# B&R Automation Studio project 8238 (part 22)

#### CmdSI.typ - BatchInformation / 1002
```iecst
(********************************************************************
 * COPYRIGHT -- Herbert Kannegiesser GmbH
 ********************************************************************
 * Library: Kanlink Cmd 1004 Status Information
 * File: CmdSI.typ
 * Author: Horn
 * Created: 02.03.2016
 ********************************************************************
 * Data types of library Kanlink
 ********************************************************************)
(*Kommando*)

TYPE
	KLreq1004_Status_typ : 	STRUCT
		wCntPositions : UINT;
		wCmdReq : UINT;
		wNoOfPosition : ARRAY[0..11]OF UINT;
	END_STRUCT;
	KLresp1004_Status_typ : 	STRUCT
		wCntPositions : UINT;
		wCmdResp : UINT;
		wNoOfPositions : ARRAY[0..11]OF UINT;
		StatusInfo : ARRAY[0..11]OF StatusInfo_typ;
	END_STRUCT;
	KL_SI_typ : 	STRUCT
		Req : KLreq1004_Status_typ;
		Resp : KLresp1004_Status_typ;
	END_STRUCT;
	StatusInfo_typ : 	STRUCT
		wStatusX : UINT;
		wSubState : UINT;
		wData1 : UINT;
		wData2 : UINT;
	END_STRUCT;
	StatusDataCmd1_typ : 	STRUCT
		wRemainCycleTime : UINT; (*Resttaktzeit bis zum Transfer*)
		wTargetCycleTime : UINT; (*Solltektzeit ohne Verkürzung oder Verlängerung*)
	END_STRUCT;
END_TYPE
```

#### CmdSilo.typ - Exported data types
```iecst
(********************************************************************
 * COPYRIGHT -- Herbert Kannegiesser GmbH
 ********************************************************************
 * Library: Kanlink
 * File: Kanlink.typ
 * Author: stahlhut
 * Created: 20.03.2012
 ********************************************************************
 * Data types of library Kanlink Commando 30010 Silo
 ********************************************************************)
(*Kommandos*)

TYPE
	KLresp30010_SH_typ : 	STRUCT
		MachineNo : STRING[15];
		State : UINT;
		RouteState : ARRAY[1..20]OF UINT;
		WetAccState : ARRAY[1..10]OF UINT;
		WetAccNiveau_mm : ARRAY[1..10]OF UINT;
		WetAccNiveau_rel : ARRAY[1..10]OF UINT;
		WetAccNiveau_Liter : ARRAY[1..10]OF UINT;
		WetAccTemp : ARRAY[1..10]OF UINT;
		WetAccMinLvlOK : ARRAY[1..10]OF UINT;
		WetAccMaxLvlOK : ARRAY[1..10]OF UINT;
	END_STRUCT;
	KLreq30010_SH_typ : 	STRUCT
		MachineNo : STRING[15];
		State : UINT;
		Handshake : BOOL;
		Route : ARRAY[1..20]OF USINT;
		TankTemp : ARRAY[1..10]OF UINT;
	END_STRUCT;
	KL_SiloData_typ : 	STRUCT
		Req : KLreq30010_SH_typ;
		Resp : KLresp30010_SH_typ;
	END_STRUCT;
END_TYPE
```

#### KLInterface.typ - Interfacetypen Kanlink
```iecst
(********************************************************************
 * COPYRIGHT -- Herbert Kannegiesser GmbH
 ********************************************************************
 * Library: Kanlink	 Interface
 * File:
 * Author: stahlhut
 * Created: 20.03.2012
 ********************************************************************
 * Data types of Interface Kanlink
 ********************************************************************)

TYPE
	KL_Key_typ : 	STRUCT
		IP_Key : UDINT;
		CmdKey : UDINT;
	END_STRUCT;
	KL_Parameter_typ : 	STRUCT
		Server : ARRAY[0..HLKANLINK_MAX_SERVERCONNS] OF KL_ServerPar_typ;
		Client : ARRAY[0..HLKANLINK_MAX_CLIENTCONNS] OF KL_ClientPar_typ;
		adrUserTyp : UDINT;
	END_STRUCT;
	KL_ClientPar_typ : 	STRUCT
		Name : STRING[15];
		Adr : UINT;
		Cmd : UINT;
		CmdOpt : UINT; (*Bits 0..3 = Nummer des Clients*)
		Area : UINT;
		CycleTime : UINT;
		sReq : STRING[80];
		sResp : STRING[80];
		AdvMode : BOOL; (*Modus mit dem eine vollständige IP-Adresse eingegeben werden kann*)
		AdrAdvMode : STRING[16]; (*Vollständige IP-Adresse*)
	END_STRUCT;
	KL_ServerPar_typ : 	STRUCT
		Name : STRING[15];
		Adr : UINT;
		Cmd : UINT;
		CmdOpt : UINT; (*Bits 0..3 = Nummer der Verbindung*)
		Area : UINT;
		TimeOut : UINT;
		sReq : STRING[80];
		sResp : STRING[80];
		AdvMode : BOOL; (*Modus mit dem eine vollständige IP-Adresse eingegeben werden kann
oder die Prüfung der IP-Adresse entfällt.*)
		AdrAdvMode : STRING[16]; (*Vollständige IP-Adresse*)
	END_STRUCT;
	IF_ServerOutTyp : 	STRUCT
		xConnected : BOOL;
		iCfgState : UINT; (*0 = ConfOK*)
		tag : UDINT;
	END_STRUCT;
	IF_Server_typ : 	STRUCT
		iState : UINT;
		out : IF_ServerOutTyp;
		tag : UDINT;
	END_STRUCT;
	IF_ClientOut_typ : 	STRUCT
		xConnected : BOOL;
		recTag : UDINT;
	END_STRUCT;
	IF_Client_typ : 	STRUCT
		out : IF_ClientOut_typ;
		iState : UINT;
		tag : UDINT;
	END_STRUCT;
	IFhlKanLink_Typ : 	STRUCT
		in : IF_KL_Control_in_typ;
		out : IF_KL_Control_out_typ;
		Server : ARRAY[0..HLKANLINK_MAX_SERVERCONNS] OF IF_Server_typ;
		Client : ARRAY[0..HLKANLINK_MAX_CLIENTCONNS] OF IF_Client_typ;
		Parameter : KL_Parameter_typ;
		xError : BOOL; (*Kanlink in Störung*)
	END_STRUCT;
	IF_KL_Control_in_typ : 	STRUCT
		xRun : BOOL; (*Rise= Starten Kanlink /fall = stoppen Kanlink*)
		xRestart : BOOL;
	END_STRUCT;
	IF_KL_Control_out_typ : 	STRUCT
		iError : UINT;
		iServerError : ARRAY[0..HLKANLINK_MAX_SERVERCONNS] OF UINT;
		iClientError : ARRAY[0..HLKANLINK_MAX_CLIENTCONNS] OF UINT;
		iStep : UINT; (*Statemachine KanLink*)
	END_STRUCT;
	IFhlKLVisuIN_typ : 	STRUCT
		cmdNr : INT; (*Ausführbares Commando*)
		cmdTag : INT; (*Dazugehörige Daten*)
		iServerNr : UINT; (*zu lesende Serverlist*)
		iCltNr : UINT; (*zu lesender Client*)
	END_STRUCT;
	IFhlKLVisuOUT_typ : 	STRUCT
		step : UINT;
		udpOpenStatus : UINT;
		udpSendStatus : UINT;
		udpRecStatus : UINT;
		iCycleTime : UINT;
		udNetId : UDINT;
		server : KL_ServerListe_typ;
		client : KL_ClientListe_typ;
		cmdResp : INT; (*Response auf CmdNr*)
	END_STRUCT;
	IFhlKLVisu_typ : 	STRUCT
		in : IFhlKLVisuIN_typ;
		out : IFhlKLVisuOUT_typ;
	END_STRUCT;
END_TYPE
```

#### KanLinkLib.typ - Exported data types
```iecst
(********************************************************************
 * COPYRIGHT -- Herbert Kannegiesser GmbH
 ********************************************************************
 * Library: WetLinkLib
 * File: WetLinkLib.typ
 * Author: stahlhut
 * Created: January 06, 2012
 ********************************************************************
 * Data types of library WetLinkLib
 ********************************************************************)
(*Interne Strukturen*)

TYPE
	udp_typ : 	STRUCT  (*UDP Typ*)
		open : UdpOpen;
		send : UdpSend;
		rec : UdpRecv;
		close : UdpClose;
	END_STRUCT;
	udint_array_typ : 	STRUCT  (*Casten von UDINT -> byte*)
		a : USINT;
		b : USINT;
		c : USINT;
		d : USINT;
	END_STRUCT;
	ServerDataTyp : 	STRUCT  (*Datatyp for global Variables*)
		receive_data : ARRAY[0..8191]OF USINT; (*Data which has been received*)
		send_data : ARRAY[0..8191]OF USINT; (*Data which should be sent*)
		PreHeaderSend : PreHeader_Typ;
		PreHeaderRec : PreHeader_Typ;
		HeaderV1Send : ARRAY[0..KLLIB_MAX_MUL]OF HeaderV1_Typ;
		HeaderV1Rec : ARRAY[0..KLLIB_MAX_MUL]OF HeaderV1_Typ;
		MetaInfoResp : KLresp0_MetaInfo_typ;
		ErrorFrame : KL_Error_Frame_typ;
		PingReq : KLreq2_Ping_typ;
		PingResp : KLresp2_Ping_typ;
		IPAdr : STRING[16]; (*IP-Adresse des Clients*)
	END_STRUCT;
	PreHeader_Typ : 	STRUCT
		Magic : UDINT; (*MagicNr*)
		HeaderVersion : UINT; (*Headerversion*)
		Tag : UINT; (*Reserve*)
	END_STRUCT;
	HeaderV1_Typ : 	STRUCT
		ReqID : UINT;
		dataFormat : UINT;
		Command : UINT;
		Length : UINT;
		CmdNr : UINT;
		CmdTag : UINT; (*Unterschiedliche Parameter zum Command*)
		Tag : UDINT; (*Reserve/Spezial*)
	END_STRUCT;
	KL_ServerListe_typ : 	STRUCT
		Cmd : UINT;
		CmdOpt : UINT;
		Adr : UINT;
		Area : UINT;
		pRespStr : UDINT; (*Adresse des Resp String*)
		pReqStr : UDINT; (*Adresse des Req String*)
		AdrDataReq : UDINT;
		ReqLength : UDINT; (*Länge Request Daten*)
		AdrDataResp : UDINT;
		RespLength : UDINT; (*Länge Response Daten*)
		Key : KL_Key_typ; (*Suchschlüssel/ Darf nicht doppelt vorkommen== Konfigurierungsfehler*)
		xConnected : BOOL; (*Falls Commando 2s nicht angefragt wird ist verbindung unterbrochen*)
		iConnectionTimer : UINT; (*Der Zugehörige Zähler / Timer*)
		adrParameter : UDINT; (*Adresse der Parameter*)
		sServerIPAdr : STRING[16];
		sClientIPAdr : STRING[16];
		iReqCnt : UINT;
		xReqManually : BOOL;
		iReqID : UINT;
		iCfgStatus : UINT;
		adrInterface : UDINT;
		xActiv : BOOL;
		tag : UDINT;
	END_STRUCT;
	KL_MuServerListe_typ : 	STRUCT
		Servers : ARRAY[0..KLLIB_MAX_MUL]OF INT;
		wOffset : ARRAY[0..KLLIB_MAX_MUL]OF UINT;
		MuServer : ARRAY[0..KLLIB_MAX_MUL]OF INT;
		lRespLength : ARRAY[0..KLLIB_MAX_MUL]OF UDINT;
		AdrRespData : ARRAY[0..KLLIB_MAX_MUL]OF UDINT;
		RespData : ARRAY[0..8191]OF USINT; (*Data which should be sent*)
		bMuServerIdx : USINT;
	END_STRUCT;
	KL_MuClientListe_typ : 	STRUCT
		bUse : USINT; (*1 = Multiclient aktiv, 2 = Multiclient wurde noch nicht geprüft, 255 = Server akzeptiert kein Multiclient*)
		Clients : ARRAY[0..KLLIB_MAX_MUL]OF INT;
		sClientAdr : STRING[16];
		iCycleTime : UINT;
		iCnt : UINT;
		iReqId : UINT;
		TimeOut : UINT;
		iTimeOutCnt : UINT;
		iCycleWait : UINT;
		xReqPending : BOOL;
		xActiv : BOOL;
		iTimeOutCnt_Summe : UINT;
		TimeOutLeft : UINT;
		xConnected : BOOL; (*True wenn Verbindung aktiv und läuft*)
		Length : UINT;
		RespLength : UDINT;
		ReqLength : UDINT;
	END_STRUCT;
	KL_ClientListe_typ : 	STRUCT
		RecCmd : UINT; (*Rec Command nr*)
		Cmd : UINT; (*Send Command nr*)
		CmdOpt : UINT; (*SendeOptionen Senden Nr des Commando etc*)
		Adr : UINT;
		Area : UINT;
		Key : KL_Key_typ;
		pResp : UDINT; (*Adresse des Namen der Response Struktur*)
		pReq : UDINT; (*Adresse des Namen der Request Struktur*)
		AdrDataReq : UDINT;
		AdrDataResp : UDINT;
		ReqLength : UDINT;
		RespLength : UDINT;
		TimeOut : UINT;
		TimeOutLeft : UINT;
		xError : BOOL;
		iCycleWait : UINT;
		iCycleTime : UINT;
		xDataRec : BOOL;
		MuClient : SINT; (*Enthalten im Multiclient*)
		iReqId : UINT;
		sClientAdr : STRING[16];
		xReqPending : BOOL;
		iTimeOutCnt : UINT;
		xActiv : BOOL;
		iCnt : UINT;
		xConnected : BOOL; (*True wenn Verbindung aktiv und läuft*)
		iTimeOutCnt_Summe : UINT;
		adrInterface : UDINT;
		adrParameter : UDINT; (*Adresse der Parameter*)
		recTag : UDINT; (*Tag des Kommandos*)
	END_STRUCT;
END_TYPE

(*Kommandos*)

TYPE
	KL_Error_Frame_typ : 	STRUCT
		Version : UINT;
		ErrorNumber : UINT;
		ErrorText : STRING[63];
	END_STRUCT;
	KLresp0_MetaInfo_typ : 	STRUCT
		KanLink_Hostname : STRING[15];
		Machine_type : STRING[15];
		SoftwareNo : STRING[15];
		SoftwareVersion : STRING[15];
		DataModelTimeStamp : DATE_AND_TIME;
		DataModelVersion : UINT;
		TimeZone : UINT;
		SommerTime : UINT;
	END_STRUCT;
	KLreq2_Ping_typ : 	STRUCT
		KanLink_Hostname : STRING[15];
	END_STRUCT;
	KLresp2_Ping_typ : 	STRUCT
		KanLink_Hostname : STRING[15];
		FrameVersion : USINT;
	END_STRUCT;
	BatchData_typ : 	STRUCT
		dtTimeStamp : DATE_AND_TIME;
		bTypeBatchNo : USINT;
		bCntCustomers : USINT;
		wTotalWeight : UINT;
		bBatchNo : ARRAY[0..15]OF USINT;
		sCategory : STRING[11];
		utfMark : ARRAY[0..31]OF UINT;
		bCustom : ARRAY[0..11]OF USINT;
		PartBatch : ARRAY[0..7]OF PartBatchData_typ;
	END_STRUCT;
	PartBatchData_typ : 	STRUCT
		sCustomNo : STRING[11];
		wCustomWeight : UINT;
	END_STRUCT;
END_TYPE
```

#### KanLinkLib.var - Exported constants
```iecst
(********************************************************************
 * COPYRIGHT -- Herbert Kannegiesser GmbH
 ********************************************************************
 * Library: WetLinkLib
 * File: WetLinkLib.var
 * Author: stahlhut
 * Created: January 06, 2012
 ********************************************************************
 * Constants of library WetLinkLib
 ********************************************************************)
VAR CONSTANT
	KLLIB_REQ : USINT := 1;
	KLLIB_MAX_MUL : USINT := 15; (*Maximale Anzahl an Clients die zusammengefasst werden dürfen*)
	KLLIB_RESP : USINT := 2;
	MagicNr : UDINT := 16#B16B00B5;
	PreHeaderSize : UDINT := 8;
	HeaderSize : UDINT := 16;
	KL_optReqManually : UINT := 16#8000;
	KL_optOnReqCall : UINT := 16#4000;
	KLLIB_MSG_NULL_POINTER : UINT := 60000;
	KLLIB_MSG_NOT_ENOUGH_MEM : UINT := 60001;
	KLLIB_MSG_VAR_ERROR : UINT := 60002;
END_VAR
```

#### KanLinkLib.fun - Exported functions and function blocks
```iecst
(********************************************************************
 * COPYRIGHT -- Herbert Kannegiesser GmbH
 ********************************************************************
 * Library: WetLinkLib
 * File: WetLinkLib.fun
 * Author: stahlhut
 * Created: January 06, 2012
 ********************************************************************
 * Functions and function blocks of library WetLinkLib
 ********************************************************************)

FUNCTION_BLOCK KanLink_FB (*TODO: Add your comment here*)
	VAR_INPUT
		Step : UINT; (*state machine*)
		ErrorNr : UINT;
		client_address : STRING[16]; (*Speichern der Receiver Adresse*)
		RecKey : KL_Key_typ;
		sNetID : STRING[15];
		udNetID : UDINT;
		udp : udp_typ;
		ServerData : ServerDataTyp;
		ServerListe : ARRAY[0..HLKANLINK_MAX_SERVERCONNS] OF KL_ServerListe_typ; (*Erlaubte Daten Server*)
		ClientListe : ARRAY[0..HLKANLINK_MAX_CLIENTCONNS] OF KL_ClientListe_typ;
		MuClientListe : ARRAY[0..HLKANLINK_MAX_MU_CLIENTCONNS] OF KL_MuClientListe_typ; (*Zusammenfasseb mehrere Clients in ein Telegramm*)
		MuServerListe : KL_MuServerListe_typ;
		_xOpenPort : BOOL;
		_xSendClient : BOOL;
		_xGetClientResp : BOOL;
		_xGetServerReq : BOOL;
		_uiLastId : UDINT;
		CanReturn : BOOL;
		adrSelf : UDINT; (*Eigene Adresse, zum weiterleiten an Function/Function Block*)
		_offset : UDINT; (*Offset zum Berechnen der Sendelänge*)
		_SendLen : UDINT; (*Sendelänge*)
		DoCommand : UINT;
		KLLib_Init_0 : KLLib_Init;
		_iCycleTime : UINT;
		adrInterface : UDINT;
		iPort : UINT; (*Port nr (23500)*)
		sIF : STRING[10]; (*Interface Ethernet*)
		CfgClient : KLLib_CfgClient;
		CfgServer : KLLib_CfgServer;
	END_VAR
	VAR_OUTPUT
		xReturn : BOOL;
	END_VAR
	VAR
		_dPrehead : REFERENCE TO PreHeader_Typ;
		_dHead : REFERENCE TO HeaderV1_Typ;
		_udArr : REFERENCE TO udint_array_typ;
		_dRecAdr : UDINT;
		_xPreheadOK : BOOL;
		_xVersionOK : BOOL;
		_xUse : BOOL;
		_i : USINT;
	END_VAR
END_FUNCTION_BLOCK

FUNCTION KLLib_ClientTimer : BOOL (*Bearbeitet Timeout und Cycletime (Zähler)*)
	VAR_INPUT
		Srv : REFERENCE TO KanLink_FB;
		_iCycleTime : UINT;
	END_VAR
	VAR
		_dClient : REFERENCE TO KL_ClientListe_typ;
		_k : UINT;
		_i : UINT;
		_dServer : REFERENCE TO KL_ServerListe_typ;
		_dInterface : REFERENCE TO IF_Client_typ;
		_dSrvIf : REFERENCE TO IF_Server_typ;
	END_VAR
END_FUNCTION

FUNCTION KLLib_GetPVAdr : UDINT (*Adresse der PV ermitteln (Server)*)
	VAR_INPUT
		ServerItem : REFERENCE TO KL_ServerListe_typ;
	END_VAR
	VAR
		iStat : INT;
	END_VAR
END_FUNCTION

FUNCTION KLLib_SendData : UDINT (*TODO: Add your comment here*)
	VAR_INPUT
		Srv : REFERENCE TO KanLink_FB;
		SendAdr : UDINT;
		SendLen : UDINT;
		pDestination : UDINT; (*Adresse des Zielstrings*)
		iIndex : INT; (*Alternativ kann zu den SendAdr und der Sende Lenge auch die Instanz des Clients angegeben werden*)
		iMuIndex : INT; (*Bei einem Multiclient wird die SendAdr und die Sende Lenge nicht angegeben.*)
		bMode : USINT; (*0 = Client; 1 = Server // Wird nur angegeben, wenn nicht die direkten Adressen angegeben werden.*)
	END_VAR
	VAR
		_i : USINT;
	END_VAR
END_FUNCTION

FUNCTION KLLib_ReadServerPara : UDINT (*TODO: Add your comment here*)
	VAR_INPUT
		adrServerItem : UDINT;
		adrParaItem : UDINT;
		adrKanLink : UDINT;
	END_VAR
	VAR
		_xError : BOOL;
		KanLink : REFERENCE TO KanLink_FB;
		dServer : REFERENCE TO KL_ServerListe_typ;
		dPara : REFERENCE TO KL_ServerPar_typ;
		_udAdr : UDINT;
		_udArr : REFERENCE TO udint_array_typ;
		_udNetId : REFERENCE TO udint_array_typ;
	END_VAR
END_FUNCTION

FUNCTION KLLib_ReadClientPara : UDINT (*TODO: Add your comment here*)
	VAR_INPUT
		adrClientItem : UDINT;
		adrParaItem : UDINT;
		adrServer : UDINT;
	END_VAR
	VAR
		_xError : BOOL;
		dClient : REFERENCE TO KL_ClientListe_typ;
		dPara : REFERENCE TO KL_ClientPar_typ;
		_udArr : REFERENCE TO udint_array_typ;
		_udAdr : UDINT;
		dServer : REFERENCE TO KanLink_FB;
		_udNetId : REFERENCE TO udint_array_typ;
	END_VAR
END_FUNCTION

FUNCTION KLLib_InitCltPV : UDINT (*TODO: Add your comment here*)
	VAR_INPUT
		dclt : REFERENCE TO KL_ClientListe_typ;
	END_VAR
	VAR
		iStat : UINT;
	END_VAR
END_FUNCTION

FUNCTION_BLOCK KLLib_Init (*TODO: Add your comment here*)
	VAR_INPUT
		enable : BOOL;
		adrServer : UDINT;
		adrInterface : UDINT;
	END_VAR
	VAR_OUTPUT
		status : UINT;
	END_VAR
	VAR
		_bStep : INT;
		_dServer : REFERENCE TO KanLink_FB;
		GetEthPort_0 : kgGetEthPort;
		CfgGetIPAddr_0 : CfgGetIPAddr;
		RTInfo_0 : RTInfo;
		_i : INT;
		_k : INT;
		_m : INT;
		_n : INT;
		_dIf : REFERENCE TO IFhlKanLink_Typ;
	END_VAR
END_FUNCTION_BLOCK

FUNCTION KL_BuildKey : BOOL
	VAR_INPUT
		Command : UINT;
		CmdNr : USINT;
		IPAdr : STRING[16];
		adrKey : UDINT;
	END_VAR
	VAR
		IP_Key : UDINT;
		Key : REFERENCE TO KL_Key_typ;
	END_VAR
END_FUNCTION

FUNCTION_BLOCK KLLib_CfgClient (*Configuriert einen Kanlink Client*)
	VAR_INPUT
		adrKanlink : UDINT;
		ClientIndex : UINT;
		adrName : UDINT;
		IPAdr : USINT;
		Area : USINT;
		CmdOpt : UINT;
		Cmd : UINT;
		CycleTime : UINT;
		adrSReq : UDINT;
		adrSResp : UDINT;
	END_VAR
	VAR_OUTPUT
		status : UINT;
	END_VAR
	VAR
		_dKL : REFERENCE TO KanLink_FB;
		_dCltPar : REFERENCE TO KL_ClientPar_typ;
		_iret : UDINT;
	END_VAR
END_FUNCTION_BLOCK

FUNCTION_BLOCK KLLib_CfgServer (*Configuriert einen Kanlink Server*)
	VAR_INPUT
		adrKanlink : UDINT;
		ServerIndex : UINT;
		adrName : UDINT;
		IPAdr : USINT;
		Area : USINT;
		CmdOpt : UINT;
		Cmd : UINT;
		TimeOut : UINT;
		adrSReq : UDINT;
		adrSResp : UDINT;
	END_VAR
	VAR_OUTPUT
		status : UINT;
	END_VAR
	VAR
		_dKL : REFERENCE TO KanLink_FB;
		_dSrvPar : REFERENCE TO KL_ServerPar_typ;
		_iret : UDINT;
	END_VAR
END_FUNCTION_BLOCK

FUNCTION KLLib_CreateStrucDef : UINT (*Erzeuge eine Strukturdefinition zu einer Variablen*)
	VAR_INPUT
		lPtrAdr : UDINT;
		lPtrLen : UDINT;
		sRootName : STRING[127];
		sItemName : STRING[31];
		lDataAdr : UDINT;
	END_VAR
	VAR
		_wStatus : UINT;
		_sPvName : STRING[127];
		_lDataType : UDINT;
		_lDataLen : UDINT;
		_wDataDimension : UINT;
		_sLine : STRING[127];
		_sValueLen : STRING[11];
		_lAdr : REFERENCE TO UDINT;
		_lLen : REFERENCE TO UDINT;
		_sValueDim : STRING[5];
		_sValueOffs : STRING[11];
		_i : UINT;
		_sItemName : STRING[31];
		_sType : ARRAY[1..23] OF STRING[15] := ['BOOL','SINT','INT','DINT','USINT','UINT','UDINT','REAL','STRING','ULINT','DATE_AND_TIME','TIME','DATE','LREAL','','TIME_OF_DAY','BYTE','WORD','DWORD','LWORD','WSTRING','','LINT'];
		_lDataAdr : UDINT;
	END_VAR
END_FUNCTION

FUNCTION KLLib_WriteStrucDefLine : UINT (*Übertrage einen String als Zeile in den Speicher*)
	VAR_INPUT
		lPtrLine : UDINT;
		lPtrAdr : UDINT;
		lPtrLen : UDINT;
	END_VAR
	VAR
		_lAdr : REFERENCE TO UDINT;
		_lLen : REFERENCE TO UDINT;
		_iStringlen : INT;
		_sLine : REFERENCE TO STRING[127];
	END_VAR
END_FUNCTION
```

#### KLLib_CfgClient.st - Configuriert einen Kanlink Client
```iecst
(********************************************************************
 * COPYRIGHT -- Herbert Kannegiesser GmbH
 ********************************************************************
 * Library: KanLinkLib
 * File: KLLib_CfgServer.st
 * Author: stahlhut
 * Created: February 01, 2012
 ********************************************************************
 * Implementation of library KanLinkLib
 ********************************************************************)

(* Configuriert einen Kanlink Client *)
FUNCTION_BLOCK KLLib_CfgClient
	// überprüfen
	IF (adrKanlink = 0) OR (adrSReq = 0) OR (adrSResp = 0) OR (adrName = 0)  THEN
		status := 1; // Fehler 1 adressen fehler
		RETURN;
	END_IF;
	IF (ClientIndex > HLKANLINK_MAX_CLIENTCONNS) THEN
		status := 2; // Fehler Index zu gross
		RETURN;
	END_IF;

	_dKL ACCESS adrKanlink;
	IF _dKL.ClientListe[ClientIndex].adrParameter = 0 THEN
		status := 3; // fehler Kanlink / fehlende init der adressen Interface
		RETURN;
	END_IF;

	IF CycleTime < 200 THEN
		CycleTime := 1000;
	END_IF;

	_dCltPar ACCESS _dKL.ClientListe[ClientIndex].adrParameter;
	_dCltPar.Adr := IPAdr;
	_dCltPar.Area := Area;
	_dCltPar.Cmd := Cmd;
	_dCltPar.CmdOpt := CmdOpt;
	memcpy(ADR( _dCltPar.Name ),adrName,15);
	memcpy(ADR(_dCltPar.sReq),adrSReq,80);
	memcpy(ADR(_dCltPar.sResp),adrSResp,80);
	_dCltPar.CycleTime := CycleTime;

	_iret := KLLib_ReadClientPara(ADR(_dKL.ClientListe[ClientIndex]),(_dKL.ClientListe[ClientIndex].adrParameter),adrKanlink);

	IF ( _iret <> 0 ) THEN
		_dKL.ClientListe[ClientIndex].xActiv := 0;
		status := 4;
	ELSE
		_dKL.ClientListe[ClientIndex].xActiv := (_dKL.ClientListe[ClientIndex].Cmd <> 0);
		status := 0; // mit ok beenden
	END_IF;

END_FUNCTION_BLOCK
```

#### KLLib_CfgServer.st - Configuriert einen Kanlink Server
```iecst
(********************************************************************
 * COPYRIGHT -- Herbert Kannegiesser GmbH
 ********************************************************************
 * Library: KanLinkLib
 * File: KLLib_CfgServer.st
 * Author: stahlhut
 * Created: February 01, 2012
 ********************************************************************
 * Implementation of library KanLinkLib
 ********************************************************************)

(* Configuriert einen Kanlink Server *)
FUNCTION_BLOCK KLLib_CfgServer
	// überprüfen
	IF (adrKanlink = 0) OR (adrSReq = 0) OR (adrSResp = 0) OR (adrName = 0)  THEN
		status := 1; // Fehler 1 adressen fehler
		RETURN;
	END_IF;
	IF (ServerIndex > HLKANLINK_MAX_SERVERCONNS) THEN
		status := 2; // Fehler Index zu gross
		RETURN;
	END_IF;

	_dKL ACCESS adrKanlink;
	IF _dKL.ServerListe[ServerIndex].adrParameter = 0 THEN
		status := 3; // fehler Kanlink / fehlende init der adressen Interface
		RETURN;
	END_IF;

	IF TimeOut < 200 THEN
		TimeOut := 1000;
	END_IF;

	_dSrvPar ACCESS _dKL.ServerListe[ServerIndex].adrParameter;
	_dSrvPar.Adr := IPAdr;
	_dSrvPar.Area := Area;
	_dSrvPar.Cmd := Cmd;
	_dSrvPar.CmdOpt := CmdOpt;
	memcpy(ADR( _dSrvPar.Name ),adrName,15);
	memcpy(ADR(_dSrvPar.sReq),adrSReq,80);
	memcpy(ADR(_dSrvPar.sResp),adrSResp,80);
	_dSrvPar.TimeOut := TimeOut;

	_iret := KLLib_ReadServerPara(ADR(_dKL.ServerListe[ServerIndex]),(_dKL.ServerListe[ServerIndex].adrParameter),adrKanlink);

	IF ( _iret <> 0 ) THEN
		status := 4;
	ELSE
		status := 0; // mit ok beenden
	END_IF;

END_FUNCTION_BLOCK
```

#### KanLink_FB.st - core-Funktion
```iecst
(********************************************************************
 * COPYRIGHT -- Herbert Kannegiesser GmbH
 ********************************************************************
 * Library: Kanlink
 * File:
 * Author: stahlhut
 * Created: January 06, 2012
 ********************************************************************
 * Implementation of library Kanlink

29.8.2012 Bug behoben verunden recAdr mit 0x0F

 ********************************************************************)

FUNCTION_BLOCK KanLink_FB

	xReturn := 0;

	IF Step <> 10 THEN
		xReturn := 1;
		RETURN;
	END_IF;
	KLLib_ClientTimer(adrSelf,_iCycleTime);

	IF  udp.send.enable THEN
		udp.send;

		IF  udp.send.status = 0 THEN
			udp.send.enable := FALSE;
		ELSIF udp.send.status = ERR_FUB_BUSY THEN
			udp.send.enable := TRUE;
			xReturn := 1;
			RETURN;
		ELSE
			ErrorNr := 4;
			udp.send.enable := FALSE;
		END_IF
	END_IF;

	udp.rec.enable := 1;
	udp.rec.ident := udp.open.ident;
	udp.rec.pData := ADR(ServerData.receive_data);	// Datenspeicher
	udp.rec.datamax := SIZEOF(ServerData.receive_data);	// Länge des Datenspeichers
	udp.rec.flags := 0;
	udp.rec.pIpAddr := ADR(client_address);	// IP Adresse des Senders
	udp.rec;

	IF udp.rec.status = 0 THEN  // Daten empfangen
		// Header Daten kopieren
		_dPrehead ACCESS ADR(ServerData.receive_data);
		_dHead ACCESS ADR(ServerData.receive_data) + PreHeaderSize;
		memcpy(ADR(ServerData.PreHeaderRec),ADR(ServerData.receive_data),PreHeaderSize);
		memset(ADR(ServerData.HeaderV1Rec),0,SIZEOF(ServerData.HeaderV1Rec));
		memcpy(ADR(ServerData.HeaderV1Rec[0]),ADR(ServerData.receive_data)+PreHeaderSize,SIZEOF(ServerData.HeaderV1Rec[0]));

		ServerData.IPAdr := client_address;

		_xPreheadOK := (ServerData.PreHeaderRec.Magic = MagicNr);
		_xVersionOK := (ServerData.PreHeaderRec.HeaderVersion = 16#100) OR (ServerData.PreHeaderRec.HeaderVersion = 16#101);

		IF (_dHead.Command AND 1) = 0 THEN
			_xGetServerReq := TRUE;
		ELSIF (_dHead.Command AND 1) = 1 THEN
			_xGetClientResp := TRUE;
		END_IF;

		IF (ServerData.PreHeaderRec.HeaderVersion = 16#101) THEN
			brsmemset(ADR(MuServerListe.wOffset),0,SIZEOF(MuServerListe.wOffset));
			brsmemset(ADR(MuServerListe.Servers),0,SIZEOF(MuServerListe.Servers));
			FOR _i := 1 TO KLLIB_MAX_MUL DO
				IF (_i = 1) THEN
					MuServerListe.wOffset[_i] := ServerData.HeaderV1Rec[_i - 1].Length + UDINT_TO_UINT(PreHeaderSize) + UDINT_TO_UINT(HeaderSize);
				ELSE
					MuServerListe.wOffset[_i] := MuServerListe.wOffset[_i - 1] + ServerData.HeaderV1Rec[_i - 1].Length + UDINT_TO_UINT(HeaderSize);
				END_IF
				IF (udp.rec.recvlen < (UINT_TO_UDINT(MuServerListe.wOffset[_i]) + HeaderSize)) THEN
					EXIT;
				END_IF
				memcpy(ADR(ServerData.HeaderV1Rec[_i]),ADR(ServerData.receive_data)+MuServerListe.wOffset[_i],SIZEOF(ServerData.HeaderV1Rec[_i]));
				IF (((ServerData.HeaderV1Rec[_i].Command = 0) AND (ServerData.HeaderV1Rec[_i].ReqID = 0)) OR ((ServerData.HeaderV1Rec[_i].Length = 0) AND (ServerData.HeaderV1Rec[_i].ReqID = 0))) THEN
					EXIT;
				END_IF
			END_FOR
		END_IF

	ELSIF udp.rec.status = udpERR_NO_DATA THEN  // Keine Daten empfangen, Client abarbeiten
		_xSendClient := TRUE;
	ELSIF udp.rec.status = ERR_FUB_BUSY THEN  (* UdpRecv not finished -> redo *)
		xReturn := 1;
		RETURN;
	ELSE  (* Goto Error Step *)
		ErrorNr := 5;
		xReturn := 1;
		RETURN;
	END_IF

	// dieser teil ist nur für den Linker (unused Variable)
	IF _xUse THEN
		_udArr;
		_dRecAdr;
		RecKey := RecKey;
		sNetID := sNetID;
		udNetID := udNetID;
		ServerListe := ServerListe;
		ClientListe	:= ClientListe;
		MuClientListe;
		_xOpenPort := _xOpenPort;
		_uiLastId	:= _uiLastId;
		CanReturn	:= CanReturn;
		_offset 	:= _offset;
		_SendLen	:= _SendLen;
		DoCommand	:= DoCommand;
	 	adrInterface	:= adrInterface;
		iPort 	:= iPort;
		sIF	:= sIF;
		KLLib_Init_0.enable	:= KLLib_Init_0.enable;
		CfgClient.adrKanlink	:= CfgClient.adrKanlink;
		CfgServer.adrKanlink	:= CfgServer.adrKanlink;
	END_IF;

END_FUNCTION_BLOCK
```

#### KLLib_ClientTimer.st
```iecst
(********************************************************************
 * COPYRIGHT -- Herbert Kannegiesser GmbH
 ********************************************************************
 * Library: WetLinkLib
 * File: WLLIb_ClientTimer.st
 * Author: stahlhut
 * Created: January 06, 2012
 ********************************************************************
 * Implementation of library WetLinkLib
 ********************************************************************)

(* TODO: Add your comment here *)
FUNCTION KLLib_ClientTimer
FOR _i := 0 TO HLKANLINK_MAX_CLIENTCONNS DO
	_dClient  ACCESS ADR(Srv.ClientListe[_i]);
	_dInterface ACCESS (_dClient.adrInterface);

	// TimeOut (kurz) taskgerecht berechnen
	IF (_dClient.TimeOutLeft >= _iCycleTime) AND _dClient.xReqPending THEN
 		_dClient.TimeOutLeft := _dClient.TimeOutLeft - _iCycleTime;
	END_IF;

	IF _dClient.iCycleWait <= _dClient.iCycleTime THEN
		_dClient.iCycleWait := _dClient.iCycleWait + _iCycleTime;
	END_IF;
	// Timeout aufgetreten nur bis n Zählen. Retry sofort nach timeout, sonst retry nach cycletime
	IF _dClient.xReqPending AND (_dClient.TimeOutLeft < _iCycleTime) THEN
		_dClient.iTimeOutCnt_Summe := _dClient.iTimeOutCnt_Summe + 1;
		_dClient.xReqPending := FALSE;	// noch mal versuchen
		IF _dClient.iTimeOutCnt < 5 THEN
			_dClient.iTimeOutCnt := _dClient.iTimeOutCnt +1 ;
			_dClient.xReqPending := FALSE;	// noch mal versuchen
			_dInterface.iState := 4;
			_dClient.iCycleWait := _dClient.iCycleTime;
		END_IF;
	END_IF;
		// Verbindungsfehler
	_dClient.xConnected := (_dClient.iTimeOutCnt < 5) AND _dClient.xActiv AND (_dClient.iCycleTime > 0);
	_dInterface.out.xConnected := _dClient.xConnected;
	IF (_dClient.iTimeOutCnt >= 5 ) AND ( _dInterface.iState = 2 ) THEN
		_dInterface.iState := 255; // Timeout melden
	END_IF;

END_FOR;

FOR _i := 0 TO HLKANLINK_MAX_MU_CLIENTCONNS DO

	// TimeOut (kurz) taskgerecht berechnen
	IF (Srv.MuClientListe[_i].TimeOutLeft >= _iCycleTime) AND Srv.MuClientListe[_i].xReqPending THEN
 		Srv.MuClientListe[_i].TimeOutLeft := Srv.MuClientListe[_i].TimeOutLeft - _iCycleTime;
	END_IF;

	IF Srv.MuClientListe[_i].iCycleWait <= Srv.MuClientListe[_i].iCycleTime THEN
		Srv.MuClientListe[_i].iCycleWait := Srv.MuClientListe[_i].iCycleWait + _iCycleTime;
	END_IF;

	// Timeout aufgetreten nur bis n Zählen. Retry sofort nach timeout, sonst retry nach cycletime
	IF Srv.MuClientListe[_i].xReqPending AND (Srv.MuClientListe[_i].TimeOutLeft < _iCycleTime) THEN
		Srv.MuClientListe[_i].iTimeOutCnt_Summe := Srv.MuClientListe[_i].iTimeOutCnt_Summe + 1;
		Srv.MuClientListe[_i].xReqPending := FALSE;	// noch mal versuchen
		IF Srv.MuClientListe[_i].iTimeOutCnt < 5 THEN
			Srv.MuClientListe[_i].iTimeOutCnt := Srv.MuClientListe[_i].iTimeOutCnt +1 ;
			Srv.MuClientListe[_i].xReqPending := FALSE;	// noch mal versuchen
			Srv.MuClientListe[_i].iCycleWait := Srv.MuClientListe[_i].iCycleTime;
		END_IF;
	END_IF;

	IF ((Srv.MuClientListe[_i].Clients[0] >= 0) AND (Srv.MuClientListe[_i].bUse <> 0) AND (Srv.MuClientListe[_i].bUse <> 255)) THEN
		FOR _k := 0 TO KLLIB_MAX_MUL DO
			IF (Srv.MuClientListe[_i].Clients[_k] >= 0) THEN
				IF (Srv.MuClientListe[_i].iCycleWait < Srv.ClientListe[Srv.MuClientListe[_i].Clients[_k]].iCycleWait) THEN
					Srv.MuClientListe[_i].iCycleWait := Srv.ClientListe[Srv.MuClientListe[_i].Clients[_k]].iCycleWait;
				END_IF
				IF (Srv.MuClientListe[_i].TimeOutLeft < Srv.ClientListe[Srv.MuClientListe[_i].Clients[_k]].TimeOutLeft) THEN
					Srv.MuClientListe[_i].TimeOutLeft := Srv.ClientListe[Srv.MuClientListe[_i].Clients[_k]].TimeOutLeft;
				END_IF
			ELSE
				EXIT;
			END_IF
		END_FOR
	ELSIF ((Srv.MuClientListe[_i].Clients[0] < 0) AND (Srv.MuClientListe[_i].bUse = 0)) THEN
		EXIT;
	END_IF
END_FOR

FOR _i := 0 TO HLKANLINK_MAX_SERVERCONNS DO
	_dServer ACCESS ADR(Srv.ServerListe[_i]);
	_dSrvIf ACCESS _dServer.adrInterface;

	IF _dServer.iConnectionTimer <= 2000 THEN
		_dServer.iConnectionTimer := _dServer.iConnectionTimer + _iCycleTime;
	END_IF;
	_dServer.xConnected := (_dServer.iConnectionTimer < 2000);
	_dSrvIf.out.xConnected := _dServer.xConnected;
END_FOR;
KLLib_ClientTimer := 0;

END_FUNCTION
```

#### KLLib_GetPVAdr.st
```iecst
(********************************************************************
 * COPYRIGHT -- Herbert Kannegiesser GmbH
 ********************************************************************
 * Library: WetLinkLib
 * File: WLLib_GetPVAdr.st
 * Author: stahlhut
 * Created: January 06, 2012
 ********************************************************************
 * Implementation of library WetLinkLib
 ********************************************************************)

(* TODO: Add your comment here *)
FUNCTION KLLib_GetPVAdr
	iStat := PV_xgetadr((ServerItem.pReqStr),ADR(ServerItem.AdrDataReq),ADR(ServerItem.ReqLength));
	IF iStat <> 0 THEN // fehler aufgetreten
 		ServerItem.AdrDataReq := 0;
		ServerItem.ReqLength := 0;
	END_IF;
	iStat := PV_xgetadr((ServerItem.pRespStr),ADR(ServerItem.AdrDataResp),ADR(ServerItem.RespLength));
	IF iStat <> 0 THEN // fehler aufgetreten
 		ServerItem.AdrDataResp := 0;
		ServerItem.RespLength := 0;
	END_IF;
	KLLib_GetPVAdr := 0;
END_FUNCTION
```

#### KLLib_SendData.st
```iecst
(********************************************************************
 * COPYRIGHT -- Herbert Kannegiesser GmbH
 ********************************************************************
 * Library: WetLinkLib
 * File: WLLib_SendData.st
 * Author: stahlhut
 * Created: January 07, 2012
 * changed April 2015
 ********************************************************************
 *
 ********************************************************************)

FUNCTION KLLib_SendData
	IF Srv.udp.send.enable = TRUE THEN //Sendung noch unterwegs, abbrechen
 		KLLib_SendData := 1;
		RETURN;
	END_IF;

	Srv.ServerData.PreHeaderSend.Magic := MagicNr;
	IF (iMuIndex >= 0) AND (bMode <> 0) THEN
		Srv.ServerData.PreHeaderSend.HeaderVersion := 16#0101;
	ELSE
		Srv.ServerData.PreHeaderSend.HeaderVersion := 16#0100;
	END_IF
	Srv._offset := 0;
	memcpy(ADR(Srv.ServerData.send_data),ADR(Srv.ServerData.PreHeaderSend),PreHeaderSize);
	Srv._offset := PreHeaderSize;

	IF (iIndex >= 0) AND (bMode <> 0) THEN
		memcpy(ADR(Srv.ServerData.send_data)+Srv._offset,ADR(Srv.ServerData.HeaderV1Send[0]),HeaderSize);
		Srv._offset := Srv._offset+ HeaderSize;
		IF (bMode <> KLLIB_REQ) THEN
			memcpy(ADR(Srv.ServerData.send_data)+Srv._offset,Srv.ClientListe[iIndex].AdrDataReq,Srv.ClientListe[iIndex].ReqLength);
		ELSIF (bMode <> KLLIB_RESP) THEN
			memcpy(ADR(Srv.ServerData.send_data)+Srv._offset,Srv.ServerListe[iIndex].AdrDataResp,Srv.ServerListe[iIndex].RespLength);
		END_IF
		Srv._SendLen := Srv._offset + Srv.ServerData.HeaderV1Send[0].Length;
	ELSIF (iMuIndex >= 0) AND (bMode = KLLIB_REQ) THEN
		Srv._SendLen := PreHeaderSize;
		FOR _i := 0 TO KLLIB_MAX_MUL DO
			IF (Srv.MuClientListe[iMuIndex].Clients[_i] >= 0) THEN
				memcpy(ADR(Srv.ServerData.send_data)+Srv._offset,ADR(Srv.ServerData.HeaderV1Send[_i]),HeaderSize);
				Srv._offset := Srv._offset + HeaderSize;
				Srv._SendLen := Srv._SendLen + HeaderSize;
				memcpy(ADR(Srv.ServerData.send_data)+Srv._offset,Srv.ClientListe[Srv.MuClientListe[iMuIndex].Clients[_i]].AdrDataReq,Srv.ClientListe[Srv.MuClientListe[iMuIndex].Clients[_i]].ReqLength);
				Srv._offset := Srv._offset+ Srv.ClientListe[Srv.MuClientListe[iMuIndex].Clients[_i]].ReqLength;
				Srv._SendLen := Srv._SendLen + Srv.ClientListe[Srv.MuClientListe[iMuIndex].Clients[_i]].ReqLength;
				Srv.MuClientListe[iMuIndex].Length := UDINT_TO_UINT(Srv._SendLen);
			ELSE
				EXIT;
			END_IF
		END_FOR
	ELSIF (iMuIndex >= 0) AND (bMode = KLLIB_RESP) THEN
		Srv._SendLen := PreHeaderSize;
		FOR _i := 0 TO KLLIB_MAX_MUL DO
			IF (Srv.MuServerListe.Servers[_i] >= 0) THEN
				memcpy(ADR(Srv.ServerData.send_data)+Srv._offset,ADR(Srv.ServerData.HeaderV1Send[_i]),HeaderSize);
				Srv._offset := Srv._offset + HeaderSize;
				Srv._SendLen := Srv._SendLen + HeaderSize;
				IF Srv.ServerData.HeaderV1Rec[_i].Command < 1000 THEN
					CASE Srv.ServerData.HeaderV1Rec[_i].Command OF
						0:   // MaschinenInfo Senden: Darf jeder lesen

							memcpy(ADR(Srv.ServerData.send_data)+Srv._offset,ADR(Srv.ServerData.MetaInfoResp),74);
							Srv._offset := Srv._offset + 74;
							Srv._SendLen := Srv._SendLen + 74;

						2:   // Response Ping: Darf jeder lesen

							memcpy(ADR(Srv.ServerData.send_data)+Srv._offset,ADR(Srv.ServerData.PingResp),17);
							Srv._offset := Srv._offset + 17;
							Srv._SendLen := Srv._SendLen + 17;

					END_CASE;

				ELSIF (Srv.MuServerListe.Servers[_i] <> 32000) THEN
					IF (Srv.MuServerListe.MuServer[_i] < 0) THEN
						memcpy(ADR(Srv.ServerData.send_data) + Srv._offset,Srv.ServerListe[Srv.MuServerListe.Servers[_i]].AdrDataResp,Srv.ServerListe[Srv.MuServerListe.Servers[_i]].RespLength);
						Srv._offset := Srv._offset + Srv.ServerListe[Srv.MuServerListe.Servers[_i]].RespLength;
						Srv._SendLen := Srv._SendLen + Srv.ServerListe[Srv.MuServerListe.Servers[_i]].RespLength;
					ELSE
						memcpy(ADR(Srv.ServerData.send_data) + Srv._offset,Srv.MuServerListe.AdrRespData[Srv.MuServerListe.MuServer[_i]],Srv.MuServerListe.lRespLength[Srv.MuServerListe.MuServer[_i]]);
						Srv._offset := Srv._offset + Srv.MuServerListe.lRespLength[Srv.MuServerListe.MuServer[_i]];
						Srv._SendLen := Srv._SendLen + Srv.MuServerListe.lRespLength[Srv.MuServerListe.MuServer[_i]];
					END_IF
				END_IF
			END_IF
		END_FOR
	ELSE
		memcpy(ADR(Srv.ServerData.send_data)+Srv._offset,ADR(Srv.ServerData.HeaderV1Send[0]),HeaderSize);
		Srv._offset := Srv._offset+ HeaderSize;
		memcpy(ADR(Srv.ServerData.send_data)+Srv._offset,SendAdr,SendLen);
		Srv._SendLen := Srv._offset + Srv.ServerData.HeaderV1Send[0].Length;
	END_IF

	// Telegramm jetzt senden
	Srv.udp.send.enable := 1;
	Srv.udp.send.ident 	:= Srv.udp.open.ident;	(* Client Ident from AsUDP.UDP_Open *)
	Srv.udp.send.pHost 	:= pDestination;	(* IP Address of the Client *)
	Srv.udp.send.port 	:= Srv.iPort;
	Srv.udp.send.pData 	:= ADR(Srv.ServerData.send_data);	(* Which data to send *)
	Srv.udp.send.datalen :=  Srv._SendLen; //
	Srv.udp.send.flags 	:= 0;
	Srv.udp.send ;	(* Call the Function*)

END_FUNCTION
```

#### KLLib_ReadServerPara.st
```iecst
(********************************************************************
 * COPYRIGHT -- Herbert Kannegiesser GmbH
 ********************************************************************
 * Library: WetLinkLib
 * File: WLLib_ReadServerPara.st
 * Author: stahlhut
 * Created: January 08, 2012
 ********************************************************************
 * Implementation of library WetLinkLib
 ********************************************************************)

(* TODO: Add your comment here *)
FUNCTION KLLib_ReadServerPara

_xError := (adrServerItem = 0) OR (adrParaItem=0) OR (adrKanLink=0);

IF _xError THEN // Fehler aufgetreten
	dServer.iCfgStatus := 2;
	KLLib_ReadServerPara := 1;
ELSE
	dServer ACCESS adrServerItem;
	dPara ACCESS adrParaItem;
	KanLink ACCESS adrKanLink;
	_udArr ACCESS ADR(_udAdr);

	dServer.iCfgStatus := 0;

	dServer.Cmd :=  dPara.Cmd;
	dServer.CmdOpt := dPara.CmdOpt;
	IF (dPara.AdvMode) THEN

	END_IF
	IF dPara.AdvMode THEN
		ethInetAton (ADR(dPara.AdrAdvMode),ADR(_udAdr));
		dServer.sServerIPAdr := dPara.AdrAdvMode;
		dServer.Area := (USINT_TO_UINT(_udArr.c) AND 16#0F);;
		dServer.Adr := USINT_TO_UINT(_udArr.d);
		dPara.Adr := dServer.Adr;
		dPara.Area := dServer.Area;
	ELSE
		dServer.Adr :=  dPara.Adr;
		dServer.Area := dPara.Area;
	END_IF
	dServer.pReqStr := ADR(dPara.sReq);
	dServer.pRespStr := ADR(dPara.sResp);
	dServer.adrParameter := adrParaItem;
	dServer.xReqManually := (dPara.CmdOpt AND KL_optReqManually) <> 0 ;
	KLLib_ReadServerPara := 0;

	_udNetId ACCESS ADR(KanLink.udNetID);
	IF NOT dPara.AdvMode THEN
		_udArr.a := _udNetId.a;
		_udArr.b := _udNetId.b;
		_udArr.c := (_udNetId.c AND 16#F0) +  UINT_TO_USINT(dServer.Area);
		_udArr.d := UINT_TO_USINT(dServer.Adr);

		ethInetNtoa((_udAdr),ADR(dServer.sServerIPAdr));
	END_IF

	KL_BuildKey(Command:= (dServer.Cmd),CmdNr := UINT_TO_USINT( dPara.CmdOpt) ,IPAdr := dServer.sServerIPAdr ,adrKey := ADR(dServer.Key));
	KLLib_GetPVAdr(adrServerItem);
	IF (dServer.AdrDataReq= 0) OR (dServer.AdrDataResp = 0) THEN
		dServer.iCfgStatus := 1; // fehler melden
	END_IF;

END_IF;

END_FUNCTION
```

#### KLLib_InitCltPV.st
```iecst
(********************************************************************
 * COPYRIGHT -- Herbert Kannegiesser GmbH
 ********************************************************************
 * Program: WetLink
 * File: WLLib_InitCltPV.st
 * Author: stahlhut
 * Created: January 06, 2012
 ********************************************************************
 * Implementation of program WetLink
 ********************************************************************)

(* TODO: Add your comment here *)
FUNCTION KLLib_InitCltPV
	iStat  := PV_xgetadr((dclt.pReq),ADR(dclt.AdrDataReq),ADR(dclt.ReqLength));
	IF iStat <> 0 THEN // fehler aufgetreten
 		dclt.AdrDataReq := 0;
		dclt.ReqLength := 0;
	END_IF;

	iStat := PV_xgetadr((dclt.pResp),ADR(dclt.AdrDataResp),ADR(dclt.RespLength));
	IF iStat <> 0 THEN // fehler aufgetreten
 		dclt.AdrDataResp := 0;
		dclt.RespLength := 0;
	END_IF;
	KLLib_InitCltPV := 0;
END_FUNCTION
```

#### KLLib_ReadClientPara.st
```iecst
(********************************************************************
 * COPYRIGHT -- Herbert Kannegiesser GmbH
 ********************************************************************
 * Library: WetLinkLib
 * File: WLLib_ReadClientPara.st
 * Author: stahlhut
 * Created: January 08, 2012
 ********************************************************************
 * Implementation of library WetLinkLib
 ********************************************************************)

(* TODO: Add your comment here *)
FUNCTION KLLib_ReadClientPara
_xError := (adrClientItem = 0) OR (adrParaItem=0) OR (adrServer = 0);

IF _xError THEN // Fehler aufgetreten
	KLLib_ReadClientPara := 1;
ELSE
	dClient ACCESS adrClientItem;
	dPara ACCESS adrParaItem;
	dServer ACCESS adrServer;
	_udArr ACCESS ADR(_udAdr);
	dClient.Cmd :=  dPara.Cmd;
	dClient.RecCmd := dPara.Cmd + 1 ;
	_udArr ACCESS ADR(_udAdr );
	IF dPara.AdvMode THEN
		ethInetAton (ADR(dPara.AdrAdvMode),(_udAdr));
		dClient.sClientAdr := dPara.AdrAdvMode;
		dClient.Area := (USINT_TO_UINT(_udArr.c) AND 16#0F);;
		dClient.Adr := USINT_TO_UINT(_udArr.d);
		dPara.Adr := dClient.Adr;
		dPara.Area := dClient.Area;
	ELSE
		dClient.Adr :=  dPara.Adr;
		dClient.Area := dPara.Area;
	END_IF
	dClient.iCycleTime := dPara.CycleTime;
	dClient.pReq := ADR(dPara.sReq);
	dClient.pResp := ADR(dPara.sResp);
	dClient.adrParameter := adrParaItem;
	dClient.CmdOpt := dPara.CmdOpt;
	KLLib_ReadClientPara := 0;

	KLLib_InitCltPV(adrClientItem);

	// Host string erzeugen

	_udNetId ACCESS ADR(dServer.udNetID);
	IF NOT dPara.AdvMode THEN
		_udArr.a := _udNetId.a;
		_udArr.b := _udNetId.b;
		_udArr.c := (_udNetId.c AND 16#F0) +  UINT_TO_USINT( dClient.Area);
		_udArr.d := UINT_TO_USINT( dClient.Adr);

		ethInetNtoa((_udAdr),ADR(dClient.sClientAdr));
	END_IF

	KL_BuildKey(Command:= dClient.RecCmd,CmdNr:=  UINT_TO_USINT(dPara.CmdOpt),IPAdr := dClient.sClientAdr, adrKey := ADR(dClient.Key));

END_IF;

END_FUNCTION
```

#### KL_BuildKey.st - Berechnen des Connection Key
```iecst
(********************************************************************
 * COPYRIGHT -- Herbert Kannegiesser GmbH
 ********************************************************************
 * Library: KanLinkLib
 * Datei: KL_BuildKey.st
 * Autor: stahlhut
 * Erstellt: 16. Januar 2012
 ********************************************************************
 * Implementierung der Library KanLinkLib
 ********************************************************************)

(* Berechnen des Connection Key *)
FUNCTION KL_BuildKey

	IF adrKey = 0 THEN // Fehler aufgetreten

		Key.CmdKey := 0;
		Key.IP_Key := 0;
		KL_BuildKey := FALSE;

	ELSE

		Key ACCESS adrKey;
		Key.CmdKey := SHL(UINT_TO_UDINT(Command),16)+USINT_TO_UINT(CmdNr);
		ethInetAton(ADR(IPAdr),ADR(IP_Key));
		Key.IP_Key := IP_Key;
		KL_BuildKey := TRUE;

	END_IF

END_FUNCTION
```

#### KLLib_Init.st
```iecst
(********************************************************************
 * COPYRIGHT -- Herbert Kannegiesser GmbH
 ********************************************************************
 * Library: KanLinkLib
 * File: KL_Init.st
 * Author: stahlhut
 * Created: January 12, 2012
 ********************************************************************
 * Implementation of library KanLinkLib
 ********************************************************************)

(* TODO: Add your comment here *)
FUNCTION_BLOCK KLLib_Init

	IF (adrServer = 0) OR (adrInterface = 0 )  THEN // fehler
		status := 1;
		enable := 0;
		RETURN;
	END_IF;
	IF enable = 0 THEN
		status := ERR_FUB_ENABLE_FALSE;
		RETURN;
	END_IF;

	IF (status = ERR_FUB_BUSY	) AND (enable = 0) THEN
		status := ERR_FUB_ENABLE_FALSE;
		_bStep := 100;
	END_IF;

	CASE _bStep OF
		0: // nix tun
			status := ERR_FUB_BUSY;
			_bStep := 10;
		10:
			_dServer ACCESS adrServer;
			_dServer.adrSelf := adrServer;
			_dIf ACCESS adrInterface;
			_dServer.adrInterface := adrInterface;

			IF _dServer.iPort = 0 THEN
				_dServer.iPort := 23500; // standardport benutzen
			END_IF;
			RTInfo_0.enable := TRUE;
			RTInfo_0;

			_dServer._iCycleTime := UDINT_TO_UINT( RTInfo_0.cycle_time / 1000);

			_bStep := 20;
		20:
			GetEthPort_0.enable := 1;
			GetEthPort_0.adrIF := ADR(_dServer.sIF);
			GetEthPort_0;
			IF GetEthPort_0.status = ERR_OK THEN
				_bStep := 30;
			ELSIF GetEthPort_0.status <> ERR_FUB_BUSY THEN // fehler aufgetreten
				status := 2;
				_bStep := 100;
			END_IF;
		30:
			CfgGetIPAddr_0.enable  := 1;
			CfgGetIPAddr_0.pDevice := ADR(_dServer.sIF);
			CfgGetIPAddr_0.pIPAddr := ADR(_dServer.sNetID);
			CfgGetIPAddr_0.Len := 16;
			CfgGetIPAddr_0;
			IF  (CfgGetIPAddr_0.status = ERR_OK) THEN
				_i := 0;
				_bStep := 40;
				ethInetAton(ADR(_dServer.sNetID),ADR(_dServer.udNetID));

			ELSIF CfgGetIPAddr_0.status <> ERR_FUB_BUSY THEN // fehler aufgetreten
				status := 3;
				_bStep := 100;
			END_IF;

		40:
			_dServer.ServerListe[_i].adrInterface := ADR(_dIf.Server[_i]);
			KLLib_ReadServerPara(ADR(_dServer.ServerListe[_i]), ADR( _dIf.Parameter.Server[_i]),ADR(_dServer));

			_i := _i + 1;
			IF (_i > HLKANLINK_MAX_SERVERCONNS) THEN
				_i := 0;
				_bStep := 41;
			END_IF

		41:
			KLLib_ReadClientPara(ADR(_dServer.ClientListe[_i]),ADR(_dIf.Parameter.Client[_i]),ADR(_dServer));
			_dServer.ClientListe[_i].xActiv := (_dServer.ClientListe[_i].Cmd <> 0);
			_dServer.ClientListe[_i].TimeOut := 140;
			_dServer.ClientListe[_i].adrInterface := ADR(_dIf.Client[_i]);
			_dServer.ClientListe[_i].MuClient := -1;

			_i := _i + 1;
			IF (_i > HLKANLINK_MAX_CLIENTCONNS) THEN
				_i := 0;
				_bStep := 45;
			END_IF

		45:
			memset(ADR(_dServer.MuClientListe),0,SIZEOF(_dServer.MuClientListe));
			FOR _m := 0 TO HLKANLINK_MAX_MU_CLIENTCONNS DO
				FOR _i := 0 TO KLLIB_MAX_MUL DO
					_dServer.MuClientListe[_m].Clients[_i] := -1;
				END_FOR
			END_FOR
			_m := 0;
			_i := 0;
			_bStep := 46;

		46:
			IF ((0 < brsstrlen(ADR(_dServer.ClientListe[_i].sClientAdr))) AND (_dServer.ClientListe[_i].Cmd <> 0)) THEN
				// Hinzufügen zu einem bestehenden Multiclient
				IF ((0 = brsstrcmp(ADR(_dServer.MuClientListe[_m].sClientAdr),ADR(_dServer.ClientListe[_i].sClientAdr))) AND (_dServer.ClientListe[_i].MuClient = -1) AND (_dServer.MuClientListe[_m].Clients[KLLIB_MAX_MUL] = -1)
					AND ((_dServer.MuClientListe[_m].ReqLength + HeaderSize + _dServer.ClientListe[_i].ReqLength) < 8192) AND ((_dServer.MuClientListe[_m].RespLength + HeaderSize + _dServer.ClientListe[_i].RespLength) < 8192)) THEN
					FOR _n := 1 TO KLLIB_MAX_MUL DO
						IF (_dServer.MuClientListe[_m].Clients[_n] = -1) THEN
							_dServer.ClientListe[_i].MuClient := INT_TO_USINT(_m);
							_dServer.MuClientListe[_m].Clients[_n] := _i;
							_dServer.MuClientListe[_m].ReqLength := _dServer.MuClientListe[_m].ReqLength + HeaderSize + _dServer.ClientListe[_i].ReqLength;
							_dServer.MuClientListe[_m].RespLength := _dServer.MuClientListe[_m].RespLength + HeaderSize + _dServer.ClientListe[_i].RespLength;
							EXIT;
						END_IF
					END_FOR
				ELSE
					FOR _k := 0 TO HLKANLINK_MAX_CLIENTCONNS DO
						// Erzeugen eines neuen MultiClients
						IF ((0 = brsstrcmp(ADR(_dServer.ClientListe[_i].sClientAdr),ADR(_dServer.ClientListe[_k].sClientAdr))) AND (_i <> _k) AND (_dServer.ClientListe[_i].MuClient = -1) AND (_dServer.ClientListe[_k].MuClient = -1) AND (_dServer.MuClientListe[_m].Clients[0] = -1)) THEN
							_dServer.MuClientListe[_m].sClientAdr := _dServer.ClientListe[_i].sClientAdr;
							_dServer.MuClientListe[_m].ReqLength := PreHeaderSize;
							_dServer.MuClientListe[_m].RespLength := PreHeaderSize;
							_dServer.ClientListe[_i].MuClient := INT_TO_USINT(_m);
							_dServer.MuClientListe[_m].Clients[0] := _i;
							_dServer.MuClientListe[_m].ReqLength := _dServer.MuClientListe[_m].ReqLength + HeaderSize + _dServer.ClientListe[_i].ReqLength;
							_dServer.MuClientListe[_m].RespLength := _dServer.MuClientListe[_m].RespLength + HeaderSize + _dServer.ClientListe[_i].RespLength;
							EXIT;
						END_IF
					END_FOR
				END_IF
			END_IF

			_i := _i + 1;
			IF (_i > HLKANLINK_MAX_CLIENTCONNS) THEN
				_i := 0;
				_m := _m + 1;
			END_IF

			IF (_m > HLKANLINK_MAX_MU_CLIENTCONNS) THEN
				_bStep := 47;
			END_IF

		47:
			// Bestimmen der Parameter für die Verbindung
			FOR _m := 0 TO HLKANLINK_MAX_MU_CLIENTCONNS DO
				IF (0 < brsstrlen(ADR(_dServer.MuClientListe[_m].sClientAdr))) THEN
					_dServer.MuClientListe[_m].bUse := 2;
					_dServer.MuClientListe[_m].TimeOut := 140;
					_dServer.MuClientListe[_m].xActiv := TRUE;
					FOR _i := 0 TO KLLIB_MAX_MUL DO
						IF (_dServer.MuClientListe[_m].Clients[_i] >= 0) THEN
							IF ((_dServer.MuClientListe[_m].iCycleTime = 0) OR ((_dServer.ClientListe[_dServer.MuClientListe[_m].Clients[_i]].iCycleTime < _dServer.MuClientListe[_m].iCycleTime) AND (_dServer.ClientListe[_dServer.MuClientListe[_m].Clients[_i]].iCycleTime > 0))) THEN
								_dServer.MuClientListe[_m].iCycleTime := _dServer.ClientListe[_dServer.MuClientListe[_m].Clients[_i]].iCycleTime;
							END_IF
						ELSE
							EXIT;
						END_IF
					END_FOR
				ELSE
					EXIT;
				END_IF
			END_FOR
			_bStep := 50;

		50:
			_dServer.udp.open.enable := 1;
			_dServer.udp.open.pIfAddr := ADR(_dServer.sNetID);	(* Übergeben des Interface funzt nicht *)
			_dServer.udp.open.port := _dServer.iPort;	(* Port to listen*)
			_dServer.udp.open.options := 0;
			_dServer.udp.open;	(* Call the Function*)

			IF _dServer.udp.open.status = 0 THEN  (* UdpOpen successful*)
				_dServer._uiLastId := _dServer.udp.open.ident;
				_bStep := 90;
			ELSIF _dServer.udp.open.status = ERR_FUB_BUSY THEN  (* UdpOpen not finished -> redo *)

			ELSIF _dServer.udp.open.status = udpERR_ALREADY_EXIST THEN // erst schliessen
				_dServer.udp.close.enable := 1;
				_dServer.udp.close.ident := _dServer._uiLastId;
				_dServer.udp.close;
				IF _dServer.udp.close.status = 0 THEN
					//
				ELSIF _dServer.udp.close.status = ERR_FUB_BUSY THEN

				ELSE
					status := 5001;
					_bStep := 100;	// unbekannter close fehler aufgetreten
				END_IF;

			ELSE
				status := 5002;
				_bStep := 100; // unbekannter open fehler aufgetreten
			END_IF

		90:  // fertig
			status := ERR_OK;
			enable := 0;
			_bStep := 0;

		100: // fehler aufgetreten
			enable := 0;
			_bStep := 0;

	END_CASE;

END_FUNCTION_BLOCK
```

#### KLLib_CreateStrucDef.st - Erzeuge eine Strukturdefinition zu einer Variablen
```iecst
(********************************************************************
 * COPYRIGHT -- Herbert Kannegiesser GmbH
 ********************************************************************
 * Library: KanLinkLib
 * File: KLLib_CreateStrucDef.st
 * Author: hunholz
 * Created: February 23, 2012
 ********************************************************************
 * Implementation of library KanLinkLib
 ********************************************************************)

(* Erzeuge eine Strukturdefinition zu einer Variablen *)

(* 1. Array müssen bei 0 beginnen
   2. Enumerationen und abgeleitete Datentypen sind verboten
*)
FUNCTION KLLib_CreateStrucDef

	KLLib_CreateStrucDef := ERR_OK;

	IF lPtrAdr = 0 OR lPtrLen = 0 THEN

		KLLib_CreateStrucDef := KLLIB_MSG_NULL_POINTER;
		RETURN;

	END_IF

	_sPvName := sRootName;

	_lAdr ACCESS lPtrAdr;
	_lLen ACCESS lPtrLen;

	IF _lAdr = 0 THEN
		KLLib_CreateStrucDef := KLLIB_MSG_NULL_POINTER;
		RETURN;
	END_IF

	IF sItemName <> '' THEN
		_sPvName := CONCAT(_sPvName, '.');
		_sPvName := CONCAT(_sPvName, sItemName);
	ELSE
		brsmemset(_lAdr, 0, _lLen);
	END_IF

	_wStatus := PV_ninfo(ADR(_sPvName), ADR(_lDataType), ADR(_lDataLen), ADR(_wDataDimension));

	IF _wStatus = ERR_OK THEN

		brsitoa(UINT_TO_DINT(_wDataDimension), ADR(_sValueDim));
		brsitoa(UDINT_TO_DINT(_lDataLen), ADR(_sValueLen));

		_wStatus := PV_xgetadr(ADR(_sPvName), ADR(_lDataAdr), ADR(_lDataLen));

		IF lDataAdr > 0 AND _lDataAdr > lDataAdr THEN

			brsitoa(UDINT_TO_DINT(_lDataAdr - lDataAdr), ADR(_sValueOffs));

		ELSE

			_sValueOffs := '0';

		END_IF

		CASE _lDataType OF

			0:  // Struktur

				_sLine := 'STRUC$T';
				_sLine := CONCAT(_sLine, sItemName);
				_sLine := CONCAT(_sLine, '$T');
				_sLine := CONCAT(_sLine, _sValueLen);
				_sLine := CONCAT(_sLine, '$T');
				_sLine := CONCAT(_sLine, _sValueOffs);
				_sLine := CONCAT(_sLine, '$T1');

				_wStatus := KLLib_WriteStrucDefLine(lPtrLine := ADR(_sLine), lPtrAdr := lPtrAdr, lPtrLen := lPtrLen);

				IF _wStatus <> ERR_OK THEN

					KLLib_CreateStrucDef := _wStatus;
					RETURN;

				END_IF

				// Die einzelnen Elemente der Struktur ermitteln

				FOR _i := 1 TO _wDataDimension DO

					_wStatus := PV_item(ADR(_sPvName), _i-1, ADR(_sItemName));

					IF _wStatus = ERR_OK THEN

						// Rekursion mit dem Strukturelement

						_wStatus := KLLib_CreateStrucDef(lPtrAdr := lPtrAdr, lPtrLen := lPtrLen, sRootName := _sPvName, sItemName := _sItemName, lDataAdr := _lDataAdr);

						IF _wStatus <> ERR_OK THEN
							KLLib_CreateStrucDef := _wStatus;
							RETURN;
						END_IF

					ELSE
						KLLib_CreateStrucDef := _wStatus;
						RETURN;
					END_IF

				END_FOR

				_sLine := 'ENDSTRUC';

				_wStatus := KLLib_WriteStrucDefLine(lPtrLine := ADR(_sLine), lPtrAdr := lPtrAdr, lPtrLen := lPtrLen);

				IF _wStatus <> ERR_OK THEN

					KLLib_CreateStrucDef := _wStatus;
					RETURN;

				END_IF

			15:	// Array einer Struktur

				_sLine := 'STRUC$T';
				_sLine := CONCAT(_sLine, sItemName);
				_sLine := CONCAT(_sLine, '$T');
				_sLine := CONCAT(_sLine, _sValueLen);
				_sLine := CONCAT(_sLine, '$T');
				_sLine := CONCAT(_sLine, _sValueOffs);
				_sLine := CONCAT(_sLine, '$T');
				_sLine := CONCAT(_sLine, _sValueDim);

				_wStatus := KLLib_WriteStrucDefLine(lPtrLine := ADR(_sLine), lPtrAdr := lPtrAdr, lPtrLen := lPtrLen);

				IF _wStatus <> ERR_OK THEN

					KLLib_CreateStrucDef := _wStatus;
					RETURN;

				END_IF

				// Um die Elemente der Struktur zu ermitteln wird PV_ninfo erneut mit einem Element des Array aufgerufen

				_sPvName := CONCAT(_sPvName,'[0]');

				_wStatus := PV_ninfo(ADR(_sPvName), ADR(_lDataType), ADR(_lDataLen), ADR(_wDataDimension));

				IF _wStatus = ERR_OK THEN

					// Die einzelnen Elemente der Struktur ermitteln

					FOR _i := 1 TO _wDataDimension DO

						_wStatus := PV_item(ADR(_sPvName), _i-1, ADR(_sItemName));

						IF _wStatus = ERR_OK THEN

							// Rekursion mit dem Strukturelement

							_wStatus := KLLib_CreateStrucDef(lPtrAdr := lPtrAdr, lPtrLen := lPtrLen, sRootName := _sPvName, sItemName := _sItemName, lDataAdr := _lDataAdr);

							IF _wStatus <> ERR_OK THEN
								KLLib_CreateStrucDef := _wStatus;
								RETURN;
							END_IF

						ELSE
							KLLib_CreateStrucDef := _wStatus;
							RETURN;
						END_IF

					END_FOR

					_sLine := 'ENDSTRUC';

					_wStatus := KLLib_WriteStrucDefLine(lPtrLine := ADR(_sLine), lPtrAdr := lPtrAdr, lPtrLen := lPtrLen);

					IF _wStatus <> ERR_OK THEN

						KLLib_CreateStrucDef := _wStatus;
						RETURN;

					END_IF

				ELSE

					KLLib_CreateStrucDef := KLLIB_MSG_VAR_ERROR;
					RETURN;

				END_IF

			1..14,16..23:

				_sLine := CONCAT(_sType[_lDataType],'$T');
				_sLine := CONCAT(_sLine, sItemName);
				_sLine := CONCAT(_sLine, '$T');
				_sLine := CONCAT(_sLine, _sValueLen);
				_sLine := CONCAT(_sLine, '$T');
				_sLine := CONCAT(_sLine, _sValueOffs);
				_sLine := CONCAT(_sLine, '$T');
				_sLine := CONCAT(_sLine, _sValueDim);

				_wStatus := KLLib_WriteStrucDefLine(lPtrLine := ADR(_sLine), lPtrAdr := lPtrAdr, lPtrLen := lPtrLen);

				IF _wStatus <> ERR_OK THEN

					KLLib_CreateStrucDef := _wStatus;
					RETURN;

				END_IF

		END_CASE

	ELSE

		KLLib_CreateStrucDef := _wStatus;
		RETURN;

	END_IF

END_FUNCTION
```

#### KLLib_WriteStrucDefLine.st - Übertrage einen String als Zeile in den Speicher
```iecst
(********************************************************************
 * COPYRIGHT -- Herbert Kannegiesser GmbH
 ********************************************************************
 * Library: KanLinkLib
 * File: KLLib_WriteStrucDefLine.st
 * Author: hunholz
 * Created: February 24, 2012
 ********************************************************************
 * Implementation of library KanLinkLib
 ********************************************************************)

(* Übertrage einen String als Zeile in den Speicher *)
FUNCTION KLLib_WriteStrucDefLine

	IF lPtrAdr = 0 OR lPtrLen = 0 OR lPtrLine = 0 THEN

		KLLib_WriteStrucDefLine := KLLIB_MSG_NULL_POINTER;
		RETURN;

	END_IF

	_lAdr ACCESS lPtrAdr;
	_lLen ACCESS lPtrLen;
	_sLine ACCESS lPtrLine;

	_sLine := CONCAT(_sLine, '$R$L');

	_iStringlen := LEN(_sLine);

	IF (INT_TO_UDINT(_iStringlen)+1) > _lLen THEN

		KLLib_WriteStrucDefLine := KLLIB_MSG_NOT_ENOUGH_MEM;
		RETURN;

	ELSE

		brsstrcpy(_lAdr, lPtrLine);
		_lAdr := _lAdr + INT_TO_UDINT(_iStringlen);
		_lLen := _lLen - INT_TO_UDINT(_iStringlen);

	END_IF

	KLLib_WriteStrucDefLine := ERR_OK;

END_FUNCTION
```

- kanlink.vsd (binary file, 171008 bytes)
### history.txt
```
1.00.7 horn	23.09.2019
Fehler behoben. In KLLib_Clinet_Timer Maximalwert für Laufvariable korrigiert.

1.00.6 horn	02.05.2019
Fehler behoben. Bei der Zusammenfassung von mehreren Client Anfragen, konnte es passieren, dass Clients gar nicht angefragt wurden.
Ein solcher Fall tritt nur dann auf, wenn mit mehreren unterschiedlichen Steuerungen kommuniziert wird.

1.00.5 horn	29.01.2019
hlKanLink kann mehrere Anfragen nach Postendaten in einem Telegramm beantworten.
Der Stand mit mehreren Clients ist für die Serie freigegeben.

1.00.4 horn	02.07.2018
hlKanLink wurde so geändert, dass mehrere Client anfragen zusammengefasst werden und in einem Telegramm zum Server geschickt werden
Der Server beantwortet die Anfragen auch wieder in einem zusammengefassten Telegramm.
Sowohl Server als auch Client seitig ist der neue KanLink kompatibel zu älteren Versionen.
Die Konstante HLKANLINK_MAX_MU_CLIENTCONNS muss in der KL_UserLib angelegt werden.
Sie bestimmt zu wie vielen Steuerungen mehrere Telegramme zusammengefasst werden dürfen. DEFAULT Empfehlung 5.

1.00.3 horn 20.03.2017
hlKanLink wurde so erweitert, dass jetzt beim Server und Client eine beliebige IP-Adresse eingegeben werden kann.
AdvMode		Freischalten der Eingabe der gesamten IP-Adresse
AdrAdvMode	gesamte IP-Adresse der Gegenstelle.

1.00.2 horn 20.01.2016
Es werden jetzt keine Warnmeldungen mehr erzeugt.

1.00.1 sta 1.4.2015 sta
KG Framework - Kompatibel
Der Client kann nun einen UDINT Tag zum Server senden. Unterstützt der Server den Tag
wird ein Server-Tag zurückgesendet.
ifhlKanlink

0.94.5 sta 16.12.2014
udp_open mit IP-Adresse binden
27.3.12/sta/Struktur für Visualisierung

20.3.12/sta/Kommando Typen in einzelne Dateien geteilt
Compiler schalter "Autonom" eingefügt, Lib Autonom erstellt
Cmd WetExt angepasst

7.3.12/sta/version Kgframework
hlKanlink Version

21.02.12 sta 0.93
Client kann mit state gesteuert werden

8.2.12 sta 0.92
Fehler bei Server-Key behoben
2.2.12 sta
Zum einrichten eines Server und Client KLLib_CfgServer und KLLib_CfgClient integriert.
Konf sowohl über Parameter und mit den Funktionen möglich

30.1.12 sta
interface  umbenannt
MaxServerConn und MaxClientCon in userlib

todo:
"OneShot" Client-Statevariable
Überprüfung Längen der Commandos
Logger wieder inbetriebnehmen

Startversion 0.900
```

### Package Logical/Standard/Kanlink/KGFrameworkShare - Benutzereinstellungen

### hlDFII.Glob.var - Package variables
```iecst
(********************************************************************
 * COPYRIGHT -- Herbert Kannegiesser GmbH
 ********************************************************************
 * File: hlDFII.Glob.var
 * Author: hunholz
 * Created: January 12, 2012
 ********************************************************************
 * Global variables of project POWERTRANSplus
 ********************************************************************)
VAR CONSTANT
	HLDFII_RUN_CLIENT : BOOL := TRUE;
	HLDFII_IDX_CPCACHE_MAX : UINT := 99;
	HLDFII_UDP_PORT_LOG4NET : UINT := 1009;
	HLDFII_MAXIDX_REQ_UPDATESTATUS : UINT := 10;
	HLDFII_MAXIDX_REQ_UPDATEBATCH : UINT := 10;
END_VAR
```

### mnCntGlob.var - Package variables
```iecst
(********************************************************************
 * COPYRIGHT -- Herbert Kannegiesser GmbH
 ********************************************************************
 * File: mnCntGlob.var
 * Author: hunholz
 * Created: November 03, 2011
 ********************************************************************
 * Global variables of project IFPOWERTRANSplusLoad
 ********************************************************************)
VAR CONSTANT
	MNCNT_MAX_RBENTRY_BATCH : UINT := 80; (*Anzahl der Einträge in der Batch-Historie*)
	MNCNT_MAX_RBENTRY_COUNTER : UINT := 500; (*Anzahl der Einträge in der Counter-Historie*)
	MNCNT_MAX_RBENTRY_TIME : UINT := 100; (*Anzahl der Einträge in der Zeit-Historie*)
	MNCNT_MAX_RBENTRY_DOSE : UINT := 1200; (*Anzahl der Einträge in der Dosierungs-Historie*)
	MNCNT_IDX_COUNTER_MAX : UINT := 127;
	MNCNT_IDX_KGMSGSTAT : UINT := 5;
END_VAR
```

### mnTxtGlob.var - Package variables
```iecst
(********************************************************************
 * COPYRIGHT -- Herbert Kannegiesser GmbH
 ********************************************************************
 * File: mnTxtGlob.var
 * Author: hunholz
 * Created: November 25, 2011
 ********************************************************************
 * Global variables of project IFPOWERTRANSplusLoad
 ********************************************************************)
(*KONSTANTEN*)
VAR CONSTANT
	MNTXT_LOAD_FUNCTIONTEXT : BOOL := TRUE; (*Lade die Funktionstexte*)
	MNTXT_LOAD_INSTANCETEXT : BOOL := TRUE; (*Lade die Instanztexte*)
	MNTXT_LOAD_PARAMETERTEXT : BOOL := TRUE; (*Lade die Parametertexte*)
	MNTXT_LOAD_PARAMTERHELPTEXT : BOOL := TRUE; (*Lade die Parameterhilfstexte*)
	MNTXT_MAX_IDX_TXT_INSTANCE : UINT := 30; (*Entsprechend der Anzahl möglicher Instanztexte*)
	MNTXT_MAX_IDX_TXT_FUNCTION : UINT := 50; (*Entsprechend der Anzahl möglicher Funktionstexte*)
	MNTXT_MAX_IDX_TXT_PARAMETER : UINT := 500; (*Entsprechend der Anzahl möglicher Parametertexte*)
END_VAR
(*Anzahl der maximal möglichen Meldungstexte kommen aus mnMsg*)
VAR CONSTANT
	MNTXT_IDX_KGMSGSTAT : UINT := 18;
	MNTXT_TEMPREADCSVSIZE : UDINT := 150000;
	MNTXT_MAXPARSELINES : UINT := 3000; (*2.000 Zeilen*)
	MNTXT_MAX_IDX_LCID : UINT := 19; (*Maximal 19 + 1 Sprache möglich*)
END_VAR
```

### mnParamGlob.var - Global variables
```iecst
(********************************************************************
 * COPYRIGHT -- Microsoft
 ********************************************************************
 * Package: --
 * File: mnParamGlob.var
 * Author: hunholz
 * Created: August 04, 2011
 ********************************************************************
 * Variables of package --
 ********************************************************************)
(*KONSTANTEN*)
VAR CONSTANT
	MNPARAM_MSGSTATIDX : UINT := 1; (*Entsprechend Zuordnungsliste*)
	MNPARAM_TEMPWRITECSVSIZE : UDINT := 75000; (*Speichergroese zum parsen von CSV-Dateien (Default: 50000)*)
	MNPARAM_MAXPARSELINES : UINT := 1500; (*Maximale Anzahl Zeilen in einer CSV-Datei inkl. Kommentare usw. Definiert die Groesse des temp. Speichers zum halten der Zeilentabelle (Default 1000)*)
	MNPARAM_CNT_LOGICSTRUCT : UINT := 150; (*Maximale Anzahl von Logical-Struct Definitionen im Datenmodell <= MNPARAM_MAXIDX_LOGICSTRUCT = 100*)
	MNPARAM_CNT_PARAMNUM : UINT := 500; (*Maximale Anzahl von numerischen Parameter Definitionen im Datenmodell <= MNPARAM_MAXIDX_PARAMNUM = 500*)
	MNPARAM_CNT_PARAMSTRING : UINT := 50; (*Maximale Anzahl von Zeichenketten Parameter Definitionen im Datenmodell <= MNPARAM_MAXIDX_PARAMSTRING = 200*)
	MNPARAM_CNT_NUMPARAMS : UINT := 5000; (*Maximale Anzahl numerischer Parameter in einem Datencontainer*)
	MNPARAM_CNT_STRINGPARAMS : UINT := 500; (*Maximale Anzahl String Parameter in einem Datencontainer*)
	MNPARAM_CNT_CSVFILES : UINT := 110; (*Maximale Anzahl möglicher CSV-Daten-Dateien*)
	MNPARAM_CNT_EDITROWS : UINT := 5; (*Anzahl der Edit-Zeilen für Parameterbearbeitung*)
	MNPARAM_CNT_NAMELIST : UINT := 100; (*Anzahl möglicher Einträge in der Namensliste für Instanzen (Programme)*)
END_VAR
(*Soll beim Importieren eines Datencontainers die Maschinennummer geprüft werden.*)
VAR CONSTANT
	MNPARAM_CMNO : UINT := 0; (*0 - Maschinennummer wird geprüft. 1 - Maschinennummer wird nicht geprüft.*)
END_VAR
(*Definition des Programmnamens*)
VAR CONSTANT
	MNPARAM_IDX_PROGCONTAINER : USINT := 2; (*Nummer des Containers mit den Programmen*)
	MNPARAM_PARIDX_PROGNAME : UINT := 4; (*Parameterindes des Stringparameters für den Programmnamen*)
END_VAR
(*Definition des Maschinennamens*)
VAR CONSTANT
	MNPARAM_IDX_MACHINENAMECONTAINER : UINT := 1; (*Nummer des Containers mit dem Maschinennamen*)
	MNPARAM_PARIDX_MACHINENAME : UINT := 5; (*Parameterindex des Stringparameters für den Maschinennamen*)
END_VAR
```

### svCPCacheGlob.var - Package variables
```iecst
(********************************************************************
 * COPYRIGHT -- Herbert Kannegiesser GmbH
 ********************************************************************
 * Package: KGFrameworkShare
 * File: svCPCacheGlob.var
 * Author: hunholz
 * Created: March 29, 2012
 ********************************************************************
 * Variables of package KGFrameworkShare
 ********************************************************************)
VAR CONSTANT
	SVCPCACHE_DB_REQUEST : USINT := 0; (*0 - keine Anfrage an der Datenbank, 1 - Anfrage bei DataFocus II*)
	SVCPCACHE_CNT_RELATIONS : UINT := 100; (*Anzahl der Kategorie-Programm-Zuordnungen*)
	SVCPCACHE_CNT_LISTRELATIONS : UINT := 10; (*Anzahl der Kategorie-Programm-Zuordnungen für die Anzeige*)
	SVCPCACHE_MAX_PARSELINES : UINT := 120; (*Maximale Anzahl von Zeilen in der CSV-Datei für die Kategorie-Programm-Relationen*)
	SVCPCACHE_NO_INDCONTAINER : USINT := 2; (*Containernummer mit Programmen*)
	SVCPCACHE_IDXPAR_NAME : UINT := 4; (*Parameterindex des Programmnamen*)
END_VAR
```

### mnSystemGlob.var - Package variables
```iecst
(********************************************************************
 * COPYRIGHT -- Herbert Kannegiesser GmbH
 ********************************************************************
 * File: mnSystemGlob.var
 * Author: hunholz
 * Created: Mar 16, 2012
 ********************************************************************
 * Global variables of project KGFramework
 ********************************************************************)
VAR CONSTANT
	MNSYSTEM_IDX_KGMSGSTAT : UINT := 102;
	MNSYSTEM_CNT_MODULELINES : UINT := 10;
	MNSYSTEM_CNT_MODULES : UINT := 10;
END_VAR
```

### Package Logical/Standard/Kanlink/KGFrameworkShare/Pkg_KGStandardShare - Projektspezifische Einstellungen

### KGStandardShare.kgMsgStatus.var - Package variables
```iecst
(********************************************************************
 * COPYRIGHT -- Microsoft
 ********************************************************************
 * Package: Pkg_KGStandardShare
 * File: KGStandardShare.kgMsgStatus.var
 * Author: hunholz
 * Created: August 25, 2011
 ********************************************************************
 * Variables of package Pkg_KGStandardShare
 ********************************************************************)
VAR CONSTANT
	MNMSG_MAX_IDX_KGMSGSTATUS : UDINT := 800; (*Anzahl der Meldequellen*)
END_VAR
```

### kgdevice.var - Package variables
```iecst
(********************************************************************
 * COPYRIGHT -- Herbert Kannegiesser GmbH
 ********************************************************************
 * Package: Pkg_KGStandard
 * File: kgdevice.var
 * Author: hunholz
 * Created: January 02, 2012
 ********************************************************************
 * Variables of package Pkg_KGStandard
 ********************************************************************)
VAR CONSTANT
	KG_DEVICE_USBSTICK1 : STRING[31] := 'USBStick1';
	KG_DEVICE_USBSTICK2 : STRING[31] := 'USBStick2';
	KG_DEVICE_COMPACTFLASH : STRING[31] := 'CFCard';
END_VAR
```

### Package Logical/Standard/Kanlink/KGFrameworkShare/Pkg_mnEthShare - Anzupassende Werte

### Pkg_mnEthShare.var - Package variables
```iecst
(********************************************************************
 * COPYRIGHT -- Microsoft
 ********************************************************************
 * Package: Pkg_mnEthShare
 * File: Pkg_mnEthShare.var
 * Author: hunholz
 * Created: June 23, 2011
 ********************************************************************
 * Variables of package Pkg_mnEthShare
 ********************************************************************)
VAR CONSTANT
	MNETH_IDX_KGMSGSTAT : UINT := 4;
END_VAR
```

### Package Logical/Standard/Kanlink/KGFrameworkShare/Pkg_mnMsgShare - Konfiguration des mnMsg

### Pkg_mnMsgShare.var - Package variables
```iecst
(********************************************************************
 * COPYRIGHT -- Microsoft
 ********************************************************************
 * Package: Pkg_mnMsgShare
 * File: Pkg_mnMsgShare.var
 * Author: hunholz
 * Created: June 21, 2011
 ********************************************************************
 * Variables of package Pkg_mnMsgShare
 ********************************************************************)
(*Globale Variable fü Meldungsmanager *)
VAR CONSTANT
	MNMSG_RUN_VC : BOOL := FALSE;
	MNMSG_MAX_IDX_VCMSGLIST : UINT := 2;
	MNMSG_MAX_IDX_VCMSGHISTLIST : UINT := 2;
	MNMSG_MAX_IDX_VCMSGSTATLIST : UINT := 2;
	MNMSG_MAX_VCMSGLISTMAINT : UINT := 1;
	MNMSG_MAX_MESSAGEHISTORY : UINT := 500; (*Anzahl der Meldungen in Ringbuffer, 500*)
	MNMSG_MAX_CFGMESSAGES : UINT := 2000; (*Anzahl der möglichen Meldungen in der Konfiguration*)
	MNMSG_IDX_KGMSGSTAT : UINT := 2;
END_VAR
```

### Package Logical/Standard/Kanlink/KGFrameworkShare/Pkg_hlKanLinkUser - Kanlink User

### Library Logical/Standard/Kanlink/KGFrameworkShare/Pkg_hlKanLinkUser/KL_UserLib (IEC, version 0.91.0) - Kanlink User Library

#### Batch.typ - Global data types
```iecst
(********************************************************************
 * COPYRIGHT --
 ********************************************************************
 * File: Batch.typ
 * Author: horn
 * Created: 01.03.2011
 * Changed: 03.08.2011
 ********************************************************************
 * Global data types of project POWERTRANSplus
 ********************************************************************)

TYPE
	BatchProcData_typ : 	STRUCT
		bProgram : USINT;
		bTypeOfLinen : USINT;
		wDisinfectionTime : UINT;
		wPreWashingTime : UINT;
		wMainWashingTime : UINT;
		wRinsingTime : UINT;
		wTotalWashingTime : UINT;
		xDrainConnectionBox : BOOL;
		xCleanConnectionBox : BOOL;
		xColorChange : BOOL;
	END_STRUCT;
	Batch_typ : 	STRUCT
		BatchData : BatchData_typ;
		BatchProcData : BatchProcData_typ;
	END_STRUCT;
	BatchLoadTrig_typ : 	STRUCT
		lTriggerChange : ARRAY[0..2] OF UDINT;
	END_STRUCT;
	BatchTrig_typ : 	STRUCT
		lTriggerChange : ARRAY[0..30] OF UDINT;
	END_STRUCT;
	BatchLoad_typ : 	STRUCT
		Batch : ARRAY[0..2] OF Batch_typ;
	END_STRUCT;
	BatchUnloadTrig_typ : 	STRUCT
		lTriggerChange : ARRAY[0..2] OF UDINT;
	END_STRUCT;
END_TYPE
```

#### KL_UserLib.typ - Exported data types
```iecst
(********************************************************************
 * COPYRIGHT -- Herbert Kannegiesser GmbH
 ********************************************************************
 * Library: WL_UserLib
 * File: WL_UserLib.typ
 * Author: stahlhut
 * Created: January 10, 2012
 ********************************************************************
 * Data types of library WL_UserLib
 ********************************************************************)

TYPE
	KL_UserTyp : 	STRUCT
		adrBatch : UDINT;
	END_STRUCT;
END_TYPE
```

#### KL_UserLib.var - Exported constants
```iecst
(********************************************************************
 * COPYRIGHT -- Herbert Kannegiesser GmbH
 ********************************************************************
 * Library: WL_UserLib
 * File: WL_UserLib.var
 * Author: stahlhut
 * Created: January 10, 2012
 ********************************************************************
 * Constants of library WL_UserLib
 ********************************************************************)
VAR CONSTANT
	HLKANLINK_MAX_CLIENTCONNS : UINT := 30; (*Anzahl der Clienten *)
	HLKANLINK_MAX_SERVERCONNS : UINT := 30; (*Anzahl der Server *)
	HLKANLINK_MAX_OVERVIEW_DATA : UINT := 31; (*Maximum data transfer on 1 overview connections*)
	HLKANLINK_MAX_MU_CLIENTCONNS : UINT := 100; (*Maximum data transfer on 1 overview connections*)
END_VAR
```

#### KL_OnRecReq.st - Wird aufgerufen bei Empfang eines Requests
```iecst
(********************************************************************
 * COPYRIGHT -- Herbert Kannegiesser GmbH
 ********************************************************************
 * Library: KL_UserLib
 * Datei: KL_OnRecReq.st
 * Autor: stahlhut
 * Erstellt: 16. Januar 2012
 ********************************************************************
 * Implementierung der Library KL_UserLib
 ********************************************************************)

(* Wird aufgerufen bei Empfang eines Requests *)
FUNCTION KL_OnRecReq
	_dKl ACCESS adrKanlink;
	s :=  _dKl.Step;

	IF (adrKanlink = 0 ) OR (adrReqData = 0) OR (adrRespData = 0) OR (adrUserData = 0) THEN
		KL_OnRecReq := 1; // fehler melden
		RETURN;
	END_IF;

	_dUserData ACCESS adrUserData;
	_dBI ACCESS  _dUserData.adrBatch;
	// Batchinfo bearbeiten
	IF iCmdNr = 1002 THEN
		_dReq ACCESS adrReqData;
		_dResp ACCESS adrRespData;

		FOR _i := 0 TO 5 DO
			IF _dReq.wNoOfPosition[_i] > 30 THEN
				_iNr := 30;
			ELSE
				_iNr := _dReq.wNoOfPosition[_i];
			END_IF;
			_dResp.BatchData[_i] :=   _dBI[_iNr].BatchData;
			_dResp.wNoOfPositions[_i] := _iNr;  //  _dReq.wNoOfPosition[_i];
		END_FOR;

	END_IF;

END_FUNCTION
```

#### KL_UserLib.fun - Exported functions and function blocks
```iecst
(********************************************************************
 * COPYRIGHT -- Herbert Kannegiesser GmbH
 ********************************************************************
 * Library: WL_UserLib
 * File: WL_UserLib.fun
 * Author: stahlhut
 * Created: January 10, 2012
 ********************************************************************
 * Functions and function blocks of library WL_UserLib
 ********************************************************************)

FUNCTION KL_OnRecReq : UDINT (*Wird aufgerufen bei Empfang eines Requests*)
	VAR_INPUT
		adrReqData : UDINT;
		adrRespData : UDINT;
		adrKanlink : UDINT;
		iCmdNr : UINT; (*Empfangene Commandnr*)
		adrUserData : UDINT;
	END_VAR
	VAR
		_dKl : REFERENCE TO KanLink_FB;
		_dResp : REFERENCE TO KLresp1002_Info_typ;
		s : INT;
		_dReq : REFERENCE TO KLreq1002_Info_typ;
		_i : UINT;
		_dUserData : REFERENCE TO KL_UserTyp;
		_dBI : REFERENCE TO ARRAY[0..30] OF Batch_typ;
		_iNr : UINT;
	END_VAR
END_FUNCTION
```

#### CmdWetExt.typ - Exported data types
```iecst
(********************************************************************
 * COPYRIGHT -- Herbert Kannegiesser GmbH
 ********************************************************************
 * Cmd 30002/Wetextraction
 * File: CmdWetExt.typ
 * Author: stahlhut
 * Created: 20.03.2012
 ********************************************************************
 * Data types of library KanlinkLib
 ********************************************************************)

TYPE
	KL_WetExtNextBatch_typ : 	STRUCT  (*Nächster Posten Entwässerung "Letzte Kammer"*)
		wProgNr : UINT;
		wWeight : UINT;
		bBatchNo : ARRAY[0..15]OF USINT;
		bTypeBatchNo : USINT;
	END_STRUCT;
	KL_WetExtRespDos_typ : 	STRUCT
		xRunning : BOOL; (*Dosierung aktiv*)
		xJobDone : BOOL; (*Dosierung beendet*)
	END_STRUCT;
	KL_WetExtReqDos_typ : 	STRUCT
		lAmount : UDINT; (*Dosiermenge für Posten*)
		xEnable : BOOL; (*Dosieren*)
	END_STRUCT;
	KL_WetExtTankInfo_typ : 	STRUCT
		wNr : UINT;
		xReady : BOOL;
		iTemperature : INT;
	END_STRUCT;
	KL_WetExtractResp_typ : 	STRUCT
		wState : UINT; (*Status der Entwässerung / nach Tis*)
		wNiveau : UINT;
		DosState : ARRAY[0..8]OF KL_WetExtRespDos_typ; (*Dosierungsstatus*)
		WetAccState : ARRAY[0..4]OF KL_WetExtTankInfo_typ;
		NextBatch : KL_WetExtNextBatch_typ;
	END_STRUCT;
	KL_WetExtractReq_typ : 	STRUCT
		wState : UINT; (*Status der Entwässerung / nach Tis*)
		wRecycleDest : UINT; (*Ziel der Rückgewinnung*)
		Dosage : ARRAY[0..8]OF KL_WetExtReqDos_typ;
		xFlush : BOOL; (*Schüttenspülung*)
		wReqTankInfo : ARRAY[0..4]OF UINT; (*Tankinfo für Nr xxx*)
		xTankReq : ARRAY[0..4]OF BOOL;
		xDrain : BOOL;
		xPump : BOOL;
		sCategory : STRING[11];
	END_STRUCT;
	KL_WetExtract_typ : 	STRUCT
		Resp : KL_WetExtractResp_typ;
		Req : KL_WetExtractReq_typ;
	END_STRUCT;
END_TYPE
```

### Package Logical/Standard/Kanlink/KGFrameworkShare/Pkg_mnTestUser - Testadapter für automatische Test

### Library Logical/Standard/Kanlink/KGFrameworkShare/Pkg_mnTestUser/libTestUse (IEC) - Userlibrary für Testadapter

#### libTestUse.typ - Exported data types
```iecst
(********************************************************************
 * COPYRIGHT -- Herbert Kannegiesser GmbH
 ********************************************************************
 * Library: libTestUse
 * File: libTestUse.typ
 * Author: hunholz
 * Created: March 06, 2012
 ********************************************************************
 * Data types of library libTestUse
 ********************************************************************)

TYPE
	TestUser_CmdTest_typ : 	STRUCT
		pCmd : ARRAY[1..LIBTEST_CNT_TSTCMD]OF UDINT;
		pParamMem : ARRAY[1..LIBTEST_CNT_TSTCMD,1..LIBTEST_CNT_TSTPARAM]OF UDINT;
		pParamSize : ARRAY[1..LIBTEST_CNT_TSTCMD,1..LIBTEST_CNT_TSTPARAM]OF UDINT;
		pCmdResult : ARRAY[1..LIBTEST_CNT_TSTCMD]OF UDINT;
		pBatchLoad : UDINT;
		pBatch : UDINT;
		pBatchUnload : UDINT;
		pBatchLoadTrig : UDINT;
		pBatchTrig : UDINT;
		pBatchUnloadTrig : UDINT;
		pBatchForLoadingOk : UDINT;
		pMachineState : UDINT;
		pMachineStateTxt : UDINT;
		pMachineStateAtt1 : UDINT;
		pMachineStateAtt2 : UDINT;
	END_STRUCT;
END_TYPE
```

#### libTest.var - Exported constants
```iecst
(********************************************************************
 * COPYRIGHT -- Herbert Kannegiesser GmbH
 ********************************************************************
 * Library: libTestUse
 * File: libTest.var
 * Author: hunholz
 * Created: March 06, 2012
 ********************************************************************
 * Constants of library libTestUse
 ********************************************************************)
VAR CONSTANT
	LIBTEST_STAT_POINTER_IS_NULL : UINT := 60000;
END_VAR
```

#### libTestUse.var - Exported constants
```iecst
(********************************************************************
 * COPYRIGHT -- Herbert Kannegiesser GmbH
 ********************************************************************
 * Library: libTestUse
 * File: libTestUse.var
 * Author: hunholz
 * Created: March 06, 2012
 ********************************************************************
 * Constants of library libTestUse
 ********************************************************************)
VAR CONSTANT
	LIBTEST_CNT_TSTCMD : UINT := 40;
	LIBTEST_CNT_TSTPARAM : UINT := 3;
END_VAR
```

#### TestUser_StopTask.st - Stoppt Task per Namen
```iecst
(********************************************************************
 * COPYRIGHT -- Herbert Kannegiesser GmbH
 ********************************************************************
 * Library: libTestUse
 * File: TestUser_StopTask.st
 * Author: hunholz
 * Created: March 06, 2012
 ********************************************************************
 * Implementation of library libTestUse
 ********************************************************************)

(* Stoppt Task per Namen *)
FUNCTION TestUser_StopTask

	TestUser_StopTask := ST_ident(st_name := st_name, st_grp := 0, st_ident := ADR(_lTaskIdent));
	IF TestUser_StopTask <> ERR_OK THEN
		RETURN;
	END_IF
	TestUser_StopTask := ST_tmp_suspend(st_ident := _lTaskIdent);

END_FUNCTION
```

#### TestUser_SetMode.st - Versetzt die Anwendung in unterschiedliche Testmodi
```iecst
(********************************************************************
 * COPYRIGHT -- Herbert Kannegiesser GmbH
 ********************************************************************
 * Library: libTestUse
 * File: TestUser_SetMode.st
 * Author: hunholz
 * Created: March 06, 2012
 ********************************************************************
 * Implementation of library libTestUse
 ********************************************************************)

(* Versetzt die Anwendung in unterschiedliche Testmodi *)
FUNCTION_BLOCK TestUser_SetMode

//	Template
//
//	IF enable THEN
//
//		IF pStruc = 0 THEN
//
//			status := LIBTEST_STAT_POINTER_IS_NULL;
//			RETURN;
//
//		ELSE
//
//			status := ERR_OK;
//
//		END_IF
//
//	ELSE
//
//		status := ERR_FUB_ENABLE_FALSE;
//
//	END_IF

	IF enable THEN

//		IF pStruc = 0 THEN
//
//			status := LIBTEST_STAT_POINTER_IS_NULL;
//			RETURN;
//
//		ELSE
//
//			status := ERR_OK;
//
		//		END_IF

		status := ERR_FUB_BUSY;

		CASE _wSetModeState OF

			0:
				status := TestUser_StopTask(st_name :=  ADR('hlKanLink'));
				IF status <> ERR_OK THEN
					RETURN;
				END_IF

				status := TestUser_StopTask(st_name :=  ADR('hlDos'));
				IF status <> ERR_OK THEN
					RETURN;
				END_IF

				status := TestUser_StopTask(st_name :=  ADR('hlSignal'));
				IF status <> ERR_OK THEN
					RETURN;
				END_IF

				status := TestUser_StopTask(st_name :=  ADR('hlDSwIn'));
				IF status <> ERR_OK THEN
					RETURN;
				END_IF

				status := TestUser_StopTask(st_name :=  ADR('hlEncode01'));
				IF status <> ERR_OK THEN
					RETURN;
				END_IF

				status := TestUser_StopTask(st_name :=  ADR('hlFC01'));
				IF status <> ERR_OK THEN
					RETURN;
				END_IF

				status := TestUser_StopTask(st_name :=  ADR('hlMotor'));
				IF status <> ERR_OK THEN
					RETURN;
				END_IF

				status := TestUser_StopTask(st_name :=  ADR('hlSafety'));
				IF status <> ERR_OK THEN
					RETURN;
				END_IF

				status := TestUser_StopTask(st_name :=  ADR('hlRate'));
				IF status <> ERR_OK THEN
					RETURN;
				END_IF

				status := TestUser_StopTask(st_name :=  ADR('hlVirtRate'));
				IF status <> ERR_OK THEN
					RETURN;
				END_IF

				status := TestUser_StopTask(st_name :=  ADR('hlValve'));
				IF status <> ERR_OK THEN
					RETURN;
				END_IF

				status := TestUser_StopTask(st_name :=  ADR('hlTemp'));
				IF status <> ERR_OK THEN
					RETURN;
				END_IF

				status := TestUser_StopTask(st_name :=  ADR('hlNiveau'));
				IF status <> ERR_OK THEN
					RETURN;
				END_IF

				status := TestUser_StopTask(st_name :=  ADR('svWetAcc'));
				IF status <> ERR_OK THEN
					RETURN;
				END_IF

				status := TestUser_StopTask(st_name :=  ADR('svRoute'));
				IF status <> ERR_OK THEN
					RETURN;
				END_IF

				status := TestUser_StopTask(st_name :=  ADR('svDrive01'));
				IF status <> ERR_OK THEN
					RETURN;
				END_IF

				status := TestUser_StopTask(st_name :=  ADR('svTakt'));
				IF status <> ERR_OK THEN
					RETURN;
				END_IF

				status := TestUser_StopTask(st_name :=  ADR('svFan'));
				IF status <> ERR_OK THEN
					RETURN;
				END_IF

				status := TestUser_StopTask(st_name :=  ADR('svCnt'));
				IF status <> ERR_OK THEN
					RETURN;
				END_IF

				status := TestUser_StopTask(st_name :=  ADR('fnWater'));
				IF status <> ERR_OK THEN
					RETURN;
				END_IF

				status := TestUser_StopTask(st_name :=  ADR('fnHeater'));
				IF status <> ERR_OK THEN
					RETURN;
				END_IF

				status := TestUser_StopTask(st_name :=  ADR('fnDrive01'));
				IF status <> ERR_OK THEN
					RETURN;
				END_IF

				status := TestUser_StopTask(st_name :=  ADR('mnComp18'));
				IF status <> ERR_OK THEN
					RETURN;
				END_IF
				status := TestUser_StopTask(st_name :=  ADR('mnComp17'));
				IF status <> ERR_OK THEN
					RETURN;
				END_IF
				status := TestUser_StopTask(st_name :=  ADR('mnComp16'));
				IF status <> ERR_OK THEN
					RETURN;
				END_IF
				status := TestUser_StopTask(st_name :=  ADR('mnComp15'));
				IF status <> ERR_OK THEN
					RETURN;
				END_IF
				status := TestUser_StopTask(st_name :=  ADR('mnComp14'));
				IF status <> ERR_OK THEN
					RETURN;
				END_IF
				status := TestUser_StopTask(st_name :=  ADR('mnComp13'));
				IF status <> ERR_OK THEN
					RETURN;
				END_IF
				status := TestUser_StopTask(st_name :=  ADR('mnComp12'));
				IF status <> ERR_OK THEN
					RETURN;
				END_IF
				status := TestUser_StopTask(st_name :=  ADR('mnComp11'));
				IF status <> ERR_OK THEN
					RETURN;
				END_IF
				status := TestUser_StopTask(st_name :=  ADR('mnComp10'));
				IF status <> ERR_OK THEN
					RETURN;
				END_IF
				status := TestUser_StopTask(st_name :=  ADR('mnComp09'));
				IF status <> ERR_OK THEN
					RETURN;
				END_IF
				status := TestUser_StopTask(st_name :=  ADR('mnComp08'));
				IF status <> ERR_OK THEN
					RETURN;
				END_IF
				status := TestUser_StopTask(st_name :=  ADR('mnComp07'));
				IF status <> ERR_OK THEN
					RETURN;
				END_IF
				status := TestUser_StopTask(st_name :=  ADR('mnComp06'));
				IF status <> ERR_OK THEN
					RETURN;
				END_IF
				status := TestUser_StopTask(st_name :=  ADR('mnComp05'));
				IF status <> ERR_OK THEN
					RETURN;
				END_IF
				status := TestUser_StopTask(st_name :=  ADR('mnComp04'));
				IF status <> ERR_OK THEN
					RETURN;
				END_IF
				status := TestUser_StopTask(st_name :=  ADR('mnComp03'));
				IF status <> ERR_OK THEN
					RETURN;
				END_IF
				status := TestUser_StopTask(st_name :=  ADR('mnComp02'));
				IF status <> ERR_OK THEN
					RETURN;
				END_IF
				status := TestUser_StopTask(st_name :=  ADR('mnComp01'));
				IF status <> ERR_OK THEN
					RETURN;
				END_IF

				status := TestUser_StopTask(st_name :=  ADR('mnTank'));
				IF status <> ERR_OK THEN
					RETURN;
				END_IF

				status := TestUser_StopTask(st_name :=  ADR('mnLoad'));
				IF status <> ERR_OK THEN
					RETURN;
				END_IF

				status := TestUser_StopTask(st_name :=  ADR('mnUnload'));
				IF status <> ERR_OK THEN
					RETURN;
				END_IF

				status := TestUser_StopTask(st_name :=  ADR('mnMaster'));
				IF status <> ERR_OK THEN
					RETURN;
				END_IF

				status := TestUser_StopTask(st_name :=  ADR('fnDos'));
				IF status <> ERR_OK THEN
					RETURN;
				END_IF

				status := TestUser_StopTask(st_name :=  ADR('hlGrease'));
				IF status <> ERR_OK THEN
					RETURN;
				END_IF

				status := TestUser_StopTask(st_name :=  ADR('hlHWCont'));
				IF status <> ERR_OK THEN
					RETURN;
				END_IF

				status := TestUser_StopTask(st_name :=  ADR('mnKanLink'));
				IF status <> ERR_OK THEN
					RETURN;
				END_IF

				status := TestUser_StopTask(st_name :=  ADR('Bufferhand'));
				IF status <> ERR_OK THEN
					RETURN;
				END_IF

				status := TestUser_StopTask(st_name :=  ADR('TestDaten'));
				IF status <> ERR_OK THEN
					RETURN;
				END_IF

				_wSetModeState := 1;
				status := ERR_OK;

			ELSE

				status := ERR_OK;

		END_CASE

	ELSE

		status := ERR_FUB_ENABLE_FALSE;
		_wSetModeState := 0;

	END_IF

END_FUNCTION_BLOCK
```

#### TestUser_RunTest.st - Zyklische Bearbeitung des Tests
```iecst
(********************************************************************
 * COPYRIGHT -- Herbert Kannegiesser GmbH
 ********************************************************************
 * Library: libTestUse
 * File: TestUser_RunTest.st
 * Author: hunholz
 * Created: March 06, 2012
 ********************************************************************
 * Implementation of library libTestUse
 ********************************************************************)

(* Zyklische Bearbeitung des Tests *)
FUNCTION_BLOCK TestUser_RunTest

//	Template
//
//	IF enable THEN
//
//		IF pStruc = 0 THEN
//
//			status := LIBTEST_STAT_POINTER_IS_NULL;
//			RETURN;
//
//		ELSE
//
//			status := ERR_OK;
//
//		END_IF
//
//	ELSE
//
//		status := ERR_FUB_ENABLE_FALSE;
//
//	END_IF

	IF enable THEN

		IF pStruc = 0 THEN

			status := KG_ERR_NULPOINTER;
			RETURN;

		END_IF

		_CmdTest ACCESS pStruc;

		status := ERR_OK;

		// Kommandos

		FOR _i := 1 TO LIBTEST_CNT_TSTCMD DO

			IF _CmdTest.pCmd[_i] = 0 THEN
				EXIT;
			ELSE
				_wCommand ACCESS _CmdTest.pCmd[_i];
			END_IF

			_bResult := 0;
			_wResult := 0;

			IF _wCommand > 0 THEN

				_bResult := kgXOR(pMem := _CmdTest.pCmd[_i] + 4, wLen := 2* SIZEOF(UDINT), bInit := _bResult, pStatus := ADR(_wXORStatus), pWordResult := ADR(_wResult));

				FOR _j := 1 TO LIBTEST_CNT_TSTPARAM DO

					IF _CmdTest.pParamMem[_i,_j] = 0 OR _CmdTest.pParamSize[_i,_j] = 0 THEN

						EXIT;

					END_IF

					_bResult := kgXOR(pMem := _CmdTest.pParamMem[_i,_j], wLen := UDINT_TO_UINT(_CmdTest.pParamSize[_i,_j]), bInit := _bResult, pStatus := ADR(_wXORStatus), pWordResult := ADR(_wResult));

				END_FOR

			END_IF

			IF _CmdTest.pCmdResult[_i] > 0 THEN

				_CmdResult ACCESS _CmdTest.pCmdResult[_i];
				_CmdResult[0] := _wResult;
				_CmdResult[1] := _wResult;

			END_IF

		END_FOR

		// Batches

		_TonShiftClck1(IN := NOT _TonShiftClck2.Q, PT := T#15s);
		_TonShiftClck2(IN := _TonShiftClck1.Q, PT := T#15s);

		IF _TonShiftClck2.Q AND _CmdTest.pBatch > 0 AND _CmdTest.pBatchLoad > 0
			AND _CmdTest.pBatchLoadTrig > 0 AND _CmdTest.pBatchTrig > 0
			AND _CmdTest.pBatchUnload > 0 AND _CmdTest.pBatchUnloadTrig > 0
			AND _CmdTest.pBatchForLoadingOk > 0 THEN

			_Batch ACCESS _CmdTest.pBatch;
			_BatchLoad ACCESS _CmdTest.pBatchLoad;
			_BatchUnload ACCESS _CmdTest.pBatchUnload;
			_BatchTrig ACCESS _CmdTest.pBatchTrig;
			_BatchLoadTrig ACCESS _CmdTest.pBatchLoadTrig;
			_BatchUnloadTrig ACCESS _CmdTest.pBatchUnloadTrig;
			_xBatchForLoadingOk ACCESS _CmdTest.pBatchForLoadingOk;

			CASE _wShiftStep OF

				0:
				// Beladeposition schreiben

					_GetTime(enable := TRUE);

					_lBatchNo := MAX(_lBatchNo+1,1);
					_pBatchNo ACCESS ADR(_BatchLoad[1].Batch[1].BatchData.bBatchNo[0]);
					_pBatchNo := _lBatchNo;

					_BatchLoad[1].Batch[1].BatchData.bCntCustomers := 1;
					_BatchLoad[1].Batch[1].BatchData.dtTimeStamp := _GetTime.DT1;

					_sValue := UDINT_TO_STRING(_lBatchNo);
					_BatchLoad[1].Batch[1].BatchData.sCategory := CONCAT('C',_sValue);
					_BatchLoad[1].Batch[1].BatchData.wTotalWeight := 300 + (UDINT_TO_UINT(_lBatchNo) MOD 1000);

					_BatchLoad[1].Batch[1].BatchData.PartBatch[0].sCustomNo := CONCAT('K',_sValue);
					_BatchLoad[1].Batch[1].BatchData.PartBatch[0].wCustomWeight := _BatchLoad[1].Batch[1].BatchData.wTotalWeight;

					_BatchLoad[2].Batch[1].BatchData := _BatchLoad[1].Batch[1].BatchData;
					_BatchLoad[3].Batch[1].BatchData := _BatchLoad[1].Batch[1].BatchData;

					_BatchLoadTrig[1].lTriggerChange[1] := _BatchLoadTrig[1].lTriggerChange[1] + 1;
					_BatchLoadTrig[2].lTriggerChange[1] := _BatchLoadTrig[2].lTriggerChange[1] + 1;
					_BatchLoadTrig[3].lTriggerChange[1] := _BatchLoadTrig[3].lTriggerChange[1] + 1;

					brsmemset(_CmdTest.pBatchUnload, 0, SIZEOF(_BatchUnload));
					_BatchUnloadTrig.lTriggerChange[1] := _BatchUnloadTrig.lTriggerChange[1] + 1;
					_BatchUnloadTrig.lTriggerChange[2] := _BatchUnloadTrig.lTriggerChange[2] + 1;

					_wShiftStep := 1;

				1:
					_Batch[0].BatchData := _BatchLoad[1].Batch[1].BatchData;
					_BatchTrig.lTriggerChange[0] := _BatchTrig.lTriggerChange[0] + 1;

					_Batch[0].BatchProcData.bProgram := UDINT_TO_USINT(_lBatchNo MOD 100);

					_xBatchForLoadingOk := TRUE;

					_wShiftStep := 2;
				2:
					_BatchUnload[1].BatchData := _Batch[30].BatchData;
					_BatchUnload[2].BatchData := _Batch[30].BatchData;
					_BatchUnloadTrig.lTriggerChange[1] := _BatchUnloadTrig.lTriggerChange[1] + 1;
					_BatchUnloadTrig.lTriggerChange[2] := _BatchUnloadTrig.lTriggerChange[2] + 1;

					FOR _j := 30 TO 2 BY -1 DO

						_Batch[_j] := _Batch[_j-1];
						_BatchTrig.lTriggerChange[_j] := _BatchTrig.lTriggerChange[_j] + 1;

					END_FOR

					brsmemset(ADR(_Batch[1]), 0, SIZEOF(_Batch[1]));
					_BatchTrig.lTriggerChange[1] := _BatchTrig.lTriggerChange[1] + 1;

					_wShiftStep := 3;
				3:

					_Batch[1] := _Batch[0];
					_BatchTrig.lTriggerChange[1] := _BatchTrig.lTriggerChange[1] + 1;

					brsmemset(ADR(_Batch[0]), 0, SIZEOF(_Batch[0]));
					_BatchTrig.lTriggerChange[0] := _BatchTrig.lTriggerChange[0] + 1;

					_xBatchForLoadingOk := FALSE;

					brsmemset(_CmdTest.pBatchLoad, 0, SIZEOF(_BatchLoad));
					_BatchLoadTrig[1].lTriggerChange[1] := _BatchLoadTrig[1].lTriggerChange[1] + 1;
					_BatchLoadTrig[2].lTriggerChange[1] := _BatchLoadTrig[2].lTriggerChange[1] + 1;
					_BatchLoadTrig[3].lTriggerChange[1] := _BatchLoadTrig[3].lTriggerChange[1] + 1;

					_wShiftStep := 0;

				ELSE

					_wShiftStep := 0;

			END_CASE

		END_IF

		// 1 s Clock

		_Ton1sClck1(IN := NOT _Ton1sClck2.Q, PT := T#500ms);
		_Ton1sClck2(IN := _Ton1sClck1.Q, PT := T#500ms);

		// MachineState

		IF _CmdTest.pMachineState > 0 AND _CmdTest.pMachineStateAtt1 > 0 AND _CmdTest.pMachineStateAtt2 > 0 AND _CmdTest.pMachineStateTxt > 0 AND _Ton1sClck2.Q THEN

			_enMachineState ACCESS _CmdTest.pMachineState;
			_wMachineStateTxt ACCESS _CmdTest.pMachineStateTxt;
			_lMachineStateAtt1 ACCESS _CmdTest.pMachineStateAtt1;
			_lMachineStateAtt2 ACCESS _CmdTest.pMachineStateAtt2;

			_wMachineStateCnt := (_wMachineStateCnt + 1) MOD 1000;

			_enMachineState := _wMachineStateCnt;
			_wMachineStateTxt := _wMachineStateCnt + 1;
			_lMachineStateAtt1 := _wMachineStateCnt + 2;
			_lMachineStateAtt2 := _wMachineStateCnt + 3;

		END_IF

	ELSE

		status := ERR_FUB_ENABLE_FALSE;

	END_IF

END_FUNCTION_BLOCK
```
